// Mitsubishi GX Works2 project: BookEX6_IP102   PLC: Q06UDV

// global labels: Global
VAR_GLOBAL
  abArray0 AT M5010 : ARRAY [0..49] OF BOOL;
  sStr0 AT D5000 : STRING[199];
  sStr1 AT D5100 : STRING[199];
  sStr2 AT D5200 : STRING[199];
  sStr3 AT D5300 : STRING[199];
  sStr4 AT D5400 : STRING[199];
  sStr5 AT D5500 : STRING[199];
  sStr6 AT D5600 : STRING[199];
  sStr7 AT D5700 : STRING[199];
  sStr8 AT D5800 : STRING[199];
  sStr9 AT D5900 : STRING[199];
  iVar0 AT D4500 : INT;
  iVar1 AT D4501 : INT;
  iVar2 AT D4502 : INT;
  iVar3 AT D4503 : INT;
  iVar4 AT D4504 : INT;
  iVar5 AT D4505 : INT;
  iVar6 AT D4506 : INT;
  iVar7 AT D4507 : INT;
  iVar8 AT D4508 : INT;
  iVar9 AT D4509 : INT;
  dVar0 AT D4510 : DINT;
  dVar1 AT D4512 : DINT;
  dVar2 AT D4514 : DINT;
  dVar3 AT D4516 : DINT;
  dVar4 AT D4518 : DINT;
  dVar5 AT D4520 : DINT;
  dVar6 AT D4522 : DINT;
  dVar7 AT D4524 : DINT;
  dVar8 AT D4526 : DINT;
  dVar9 AT D4528 : DINT;
  wVar0 AT D4530 : WORD;
  wVar1 AT D4531 : WORD;
  wVar2 AT D4532 : WORD;
  wVar3 AT D4533 : WORD;
  wVar4 AT D4534 : WORD;
  wVar5 AT D4535 : WORD;
  wVar6 AT D4536 : WORD;
  wVar7 AT D4537 : WORD;
  wVar8 AT D4538 : WORD;
  wVar9 AT D4539 : WORD;
  dwVar0 AT D4540 : DWORD;
  dwVar1 AT D4542 : DWORD;
  dwVar2 AT D4544 : DWORD;
  dwVar3 AT D4546 : DWORD;
  dwVar4 AT D4548 : DWORD;
  dwVar5 AT D4550 : DWORD;
  dwVar6 AT D4552 : DWORD;
  dwVar7 AT D4554 : DWORD;
  dwVar8 AT D4556 : DWORD;
  dwVar9 AT D4558 : DWORD;
  fsVar0 AT D4560 : REAL;
  fsVar1 AT D4562 : REAL;
  fsVar2 AT D4564 : REAL;
  fsVar3 AT D4566 : REAL;
  fsVar4 AT D4568 : REAL;
  fsVar5 AT D4570 : REAL;
  fsVar6 AT D4572 : REAL;
  fsVar7 AT D4574 : REAL;
  fsVar8 AT D4576 : REAL;
  fsVar9 AT D4578 : REAL;
  fdVar0 AT D4580 : LREAL;
  tTime0 AT D4620 : TIME;
  tTime1 AT D4622 : TIME;
  tTime2 AT D4624 : TIME;
  tTime3 AT D4626 : TIME;
  tTime4 AT D4628 : TIME;
  tTime5 AT D4630 : TIME;
  tTime6 AT D4632 : TIME;
  tTime7 AT D4634 : TIME;
  tTime8 AT D4636 : TIME;
  tTime9 AT D4638 : TIME;
  tTime10 AT D4640 : TIME;
  bVar1 AT M5001 : BOOL;
  bVar2 AT M5002 : BOOL;
  bVar3 AT M5003 : BOOL;
  bVar4 AT M5004 : BOOL;
  bVar5 AT M5005 : BOOL;
  bVar6 AT M5006 : BOOL;
  bVar7 AT M5007 : BOOL;
  bVar8 AT M5008 : BOOL;
  bVar9 AT M5009 : BOOL;
  abArray1 AT M5060 : ARRAY [0..49] OF BOOL;
  abArray2 AT M5110 : ARRAY [0..49] OF BOOL;
  abArray3 AT M5160 : ARRAY [0..49] OF BOOL;
  abArray4 AT M5210 : ARRAY [0..49] OF BOOL;
  abArray5 AT M5260 : ARRAY [0..49] OF BOOL;
  abArray6 AT M5310 : ARRAY [0..49] OF BOOL;
  abArray7 AT M5360 : ARRAY [0..49] OF BOOL;
  abArray8 AT M5410 : ARRAY [0..49] OF BOOL;
  abArray9 AT M5460 : ARRAY [0..49] OF BOOL;
  fdVar1 AT D4584 : LREAL;
  fdVar2 AT D4588 : LREAL;
  fdVar3 AT D4592 : LREAL;
  fdVar4 AT D4596 : LREAL;
  fdVar5 AT D4600 : LREAL;
  fdVar6 AT D4604 : LREAL;
  fdVar7 AT D4608 : LREAL;
  fdVar8 AT D4612 : LREAL;
  fdVar9 AT D4616 : LREAL;
  bVar0 AT M5000 : BOOL;
END_VAR

// global labels: QPLCSpecial
VAR_GLOBAL
  sbGetTime AT SM213 : BOOL;
  sbOn AT SM400 : BOOL;
  sbOff AT SM401 : BOOL;
  sbOn1Time AT SM402 : BOOL;
  sbOff1Time AT SM403 : BOOL;
  sb5ms AT SM409 : BOOL;
  sdSwitch AT SD200 : INT;
  sdTime03 AT SD212 : INT;
  sdTime04 AT SD213 : INT;
  sdTime02 AT SD211 : INT;
  sdTime01 AT SD210 : INT;
  sdScanTime1 AT SD521 : INT;
  sdScanTimeMin1 AT SD525 : INT;
  sdScanTimeMin AT SD524 : INT;
  sdScanTimeMax1 AT SD527 : INT;
  sdScanTimeMax AT SD526 : INT;
  sbErrInfo2 AT SM16 : BOOL;
  sbErrInfo AT SM5 : BOOL;
  sbSelfError AT SM1 : BOOL;
  sbDiagError AT SM0 : BOOL;
  sbResetErr AT SM50 : BOOL;
  sbSetTime AT SM210 : BOOL;
  sbFuse AT SM60 : BOOL;
  sbOpError AT SM56 : BOOL;
  sbPowerDown AT SM53 : BOOL;
  sbBatLow AT SM52 : BOOL;
  sbBatLowL AT SM51 : BOOL;
  sbSTOP AT SM203 : BOOL;
  sbPAUSE AT SM204 : BOOL;
  sbNsec AT SM414 : BOOL;
  sb1000ms AT SM413 : BOOL;
  sb500ms AT SM412 : BOOL;
  sbNms AT SM415 : BOOL;
  sbUserClk4 AT SM424 : BOOL;
  sbUserClk3 AT SM423 : BOOL;
  sbUserClk2 AT SM422 : BOOL;
  sbUserClk1 AT SM421 : BOOL;
  sbUserClk0 AT SM420 : BOOL;
  sdBatLowL AT SD51 : INT;
  sdPLCErrInfo AT SD4 : INT;
  sdPLCErrDate2 AT SD3 : INT;
  sdPLCErrDate1 AT SD2 : INT;
  sdPLCErrDate0 AT SD1 : INT;
  sdPLCErrCode AT SD0 : INT;
  sdFuse AT SD60 : INT;
  sdPowerDown AT SD53 : INT;
  sdBatLow AT SD52 : INT;
  sdCPUSts AT SD203 : INT;
  sdLed AT SD201 : INT;
  sdScanTime AT SD520 : INT;
  sdCntNsec AT SD414 : INT;
  sdCnt1sec AT SD412 : INT;
  sdCntScan AT SD420 : INT;
  sdCntNms AT SD415 : INT;
  sb100ms AT SM411 : BOOL;
  sb50ms AT SM410 : BOOL;
  sdSckOpenComp AT SD1282 : WORD;
  sdSckOpenReq AT SD1284 : WORD;
  sdSckDataRx AT SD1286 : WORD;
  sdSckConn AT SD1288 : WORD;
END_VAR

// global labels: Network
VAR_GLOBAL
  aSendData1 AT D100 : ARRAY [0..4] OF INT;
  aiTxData AT D4000 : ARRAY [0..99] OF INT;
  aiRxData AT D4100 : ARRAY [0..99] OF INT;
  iOpenOK AT D3900 : INT;
  iOpenERR AT D3901 : INT;
  iSendOK AT D3902 : INT;
  iSendERR AT D3903 : INT;
  iCloseOK AT D3906 : INT;
  iCloseERR AT D3907 : INT;
  iRecvOK AT D3904 : INT;
  iRecvERR AT D3905 : INT;
  aiTxData2 AT D4200 : ARRAY [0..99] OF INT;
  aiRxData2 AT D4300 : ARRAY [0..99] OF INT;
  iOpenOK2 AT D3908 : INT;
  iOpenERR2 AT D3909 : INT;
  iSendOK2 AT D3910 : INT;
  iSendERR2 AT D3911 : INT;
  iRecvOK2 AT D3912 : INT;
  iRecvERR2 AT D3913 : INT;
  iCloseOK2 AT D3914 : INT;
  iCloseERR2 AT D3915 : INT;
  iEOpenComp AT D3916 : INT;
  iEOpenReq AT D3917 : INT;
  iERecvFlag AT D3918 : INT;
  iOpenCode AT D3919 : INT;
  iSendCode AT D3920 : INT;
  iRecvCode AT D3921 : INT;
  iCloseCode AT D3922 : INT;
  iOpenCode2 AT D3923 : INT;
  iSendCode2 AT D3924 : INT;
  iRecvCode2 AT D3925 : INT;
  iCloseCode2 AT D3926 : INT;
  aRecvData1 AT D105 : ARRAY [0..4] OF INT;
  aSendData2 AT D110 : ARRAY [0..4] OF INT;
  aRecvData2 AT D115 : ARRAY [0..4] OF INT;
  aSendData3 AT D120 : ARRAY [0..4] OF INT;
  aRecvData3 AT D125 : ARRAY [0..4] OF INT;
  aRdata AT D140 : ARRAY [0..9] OF INT;
  aSLMPDataTx AT D150 : ARRAY [0..9] OF WORD;
  aSLMPDataRx AT D160 : ARRAY [0..9] OF WORD;
END_VAR
// user libraries (not included): HMI

PROGRAM ExUINI
VAR
  bReq : BOOL;
  Mov8INT_1 : Mov8INT;
  abComp : ARRAY [0..1] OF BOOL;
  bNormal : BOOL;
  bError : BOOL;
END_VAR
(* structured ladder/FBD written out as ST: instructions are called as NAME(EN, inputs, outputs); _pN, _eN, _tN stand for wires *)
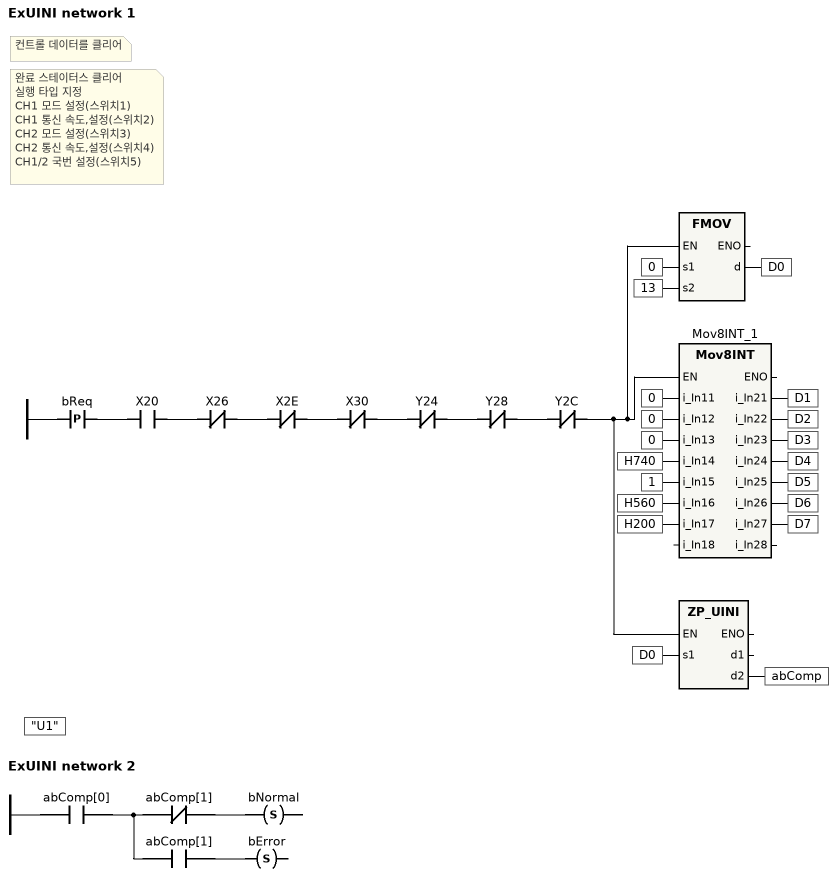
(* network 1 *)
(* 컨트롤 데이터를 클리어 *)
(* 완료 스테이터스 클리어 / 실행 타입 지정 / CH1 모드 설정(스위치1) / CH1 통신 속도,설정(스위치2) / CH2 모드 설정(스위치3) / CH2 통신 속도,설정(스위치4) / CH1/2 국번 설정(스위치5) *)
_p1 := LDP(TRUE, bReq) AND X20 AND NOT X26 AND NOT X2E AND NOT X30 AND NOT Y24 AND NOT Y28 AND NOT Y2C;
FMOV(_p1, 0, 13, D0);
Mov8INT_1(EN := _p1, i_In11 := 0, i_In12 := 0, i_In13 := 0, i_In14 := H740, i_In15 := 1, i_In16 := H560, i_In17 := H200, i_In21 => D1, i_In22 => D2, i_In23 => D3, i_In24 => D4, i_In25 => D5, i_In26 => D6, i_In27 => D7);
ZP_UINI(_p1, D0, _open, abComp);
(* not connected to any output: "U1" *)
(* network 2 *)
SET(abComp[0] AND NOT abComp[1], bNormal);
SET(abComp[0] AND abComp[1], bError);
END_PROGRAM

PROGRAM Ez_ethREAD_WRITE
VAR
  Mov8INT_1 : Mov8INT;
  acRdCtrl : ARRAY [0..17] OF INT;
  abRdComp : ARRAY [0..1] OF BOOL;
  iCntRdOk : INT;
  iCntRdErr : INT;
END_VAR
(* structured ladder/FBD written out as ST: instructions are called as NAME(EN, inputs, outputs); _pN, _eN, _tN stand for wires *)
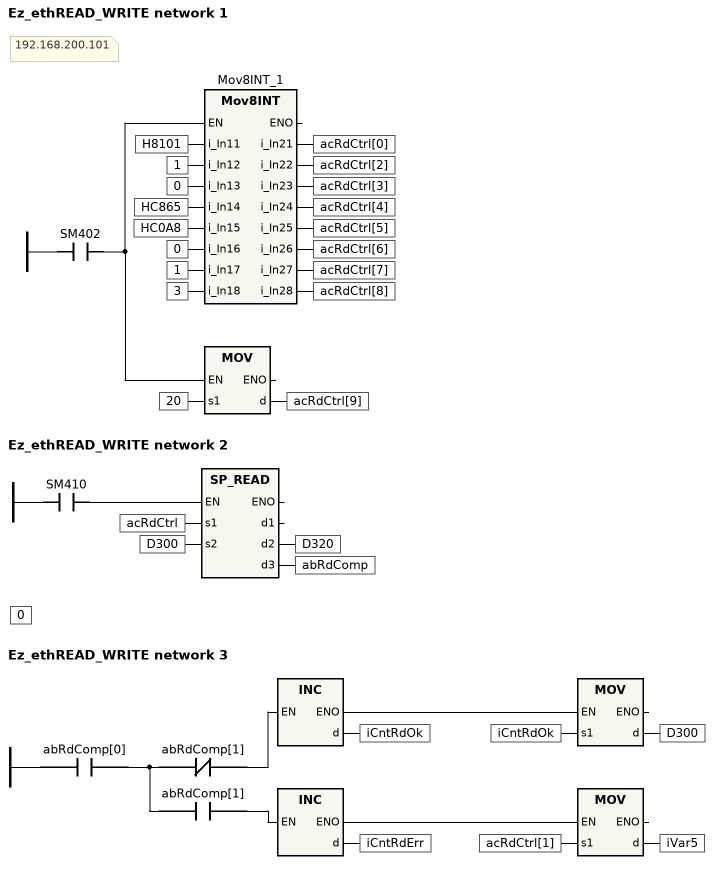
(* network 1 *)
(* 192.168.200.101 *)
Mov8INT_1(EN := SM402, i_In11 := H8101, i_In12 := 1, i_In13 := 0, i_In14 := HC865, i_In15 := HC0A8, i_In16 := 0, i_In17 := 1, i_In18 := 3, i_In21 => acRdCtrl[0], i_In22 => acRdCtrl[2], i_In23 => acRdCtrl[3], i_In24 => acRdCtrl[4], i_In25 => acRdCtrl[5], i_In26 => acRdCtrl[6], i_In27 => acRdCtrl[7], i_In28 => acRdCtrl[8]);
MOV(SM402, 20, acRdCtrl[9]);
(* network 2 *)
SP_READ(SM410, acRdCtrl, D300, _open, D320, abRdComp);
(* not connected to any output: 0 *)
(* network 3 *)
_e1 := INC(abRdComp[0] AND NOT abRdComp[1], iCntRdOk);
MOV(_e1, iCntRdOk, D300);
_e2 := INC(abRdComp[0] AND abRdComp[1], iCntRdErr);
MOV(_e2, acRdCtrl[1], iVar5);
END_PROGRAM

PROGRAM ExSample
VAR
  Mov8INT_1 : Mov8INT;
  Mov8INT_2 : Mov8INT;
  Mov8INT_3 : Mov8INT;
  Mov8INT_4 : Mov8INT;
  Mov8INT_5 : Mov8INT;
  Mov8INT_6 : Mov8INT;
END_VAR
(* structured ladder/FBD written out as ST: instructions are called as NAME(EN, inputs, outputs); _pN, _eN, _tN stand for wires *)
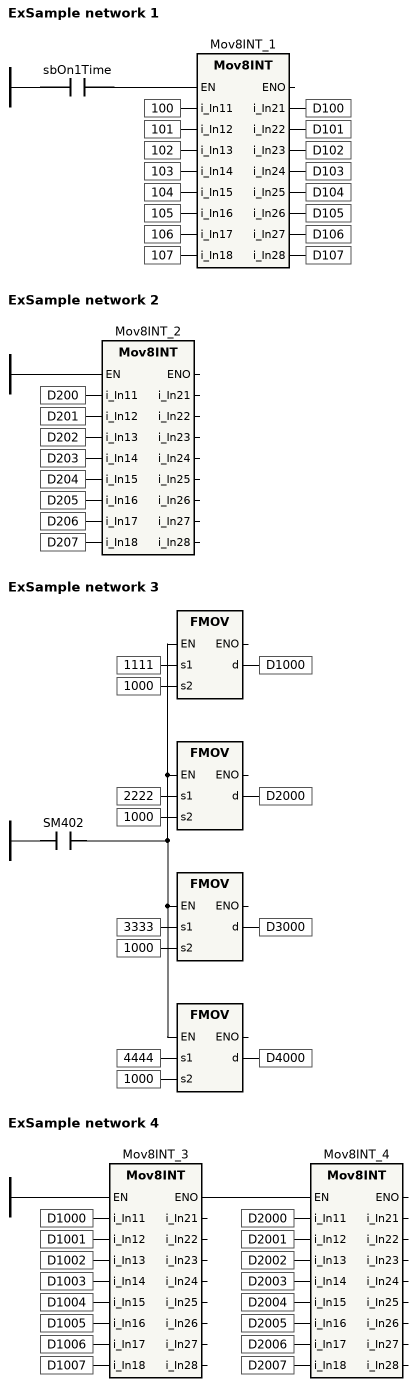
(* network 1 *)
Mov8INT_1(EN := sbOn1Time, i_In11 := 100, i_In12 := 101, i_In13 := 102, i_In14 := 103, i_In15 := 104, i_In16 := 105, i_In17 := 106, i_In18 := 107, i_In21 => D100, i_In22 => D101, i_In23 => D102, i_In24 => D103, i_In25 => D104, i_In26 => D105, i_In27 => D106, i_In28 => D107);
(* network 2 *)
Mov8INT_2(EN := TRUE, i_In11 := D200, i_In12 := D201, i_In13 := D202, i_In14 := D203, i_In15 := D204, i_In16 := D205, i_In17 := D206, i_In18 := D207);
(* network 3 *)
FMOV(SM402, 1111, 1000, D1000);
FMOV(SM402, 2222, 1000, D2000);
FMOV(SM402, 3333, 1000, D3000);
FMOV(SM402, 4444, 1000, D4000);
(* network 4 *)
Mov8INT_3(EN := TRUE, i_In11 := D1000, i_In12 := D1001, i_In13 := D1002, i_In14 := D1003, i_In15 := D1004, i_In16 := D1005, i_In17 := D1006, i_In18 := D1007);
Mov8INT_4(EN := Mov8INT_3.ENO, i_In11 := D2000, i_In12 := D2001, i_In13 := D2002, i_In14 := D2003, i_In15 := D2004, i_In16 := D2005, i_In17 := D2006, i_In18 := D2007);
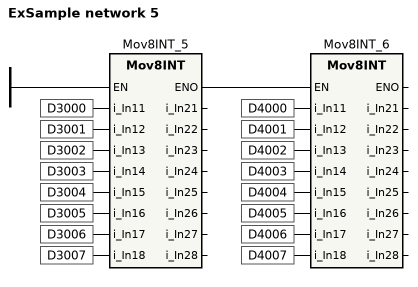
(* network 5 *)
Mov8INT_5(EN := TRUE, i_In11 := D3000, i_In12 := D3001, i_In13 := D3002, i_In14 := D3003, i_In15 := D3004, i_In16 := D3005, i_In17 := D3006, i_In18 := D3007);
Mov8INT_6(EN := Mov8INT_5.ENO, i_In11 := D4000, i_In12 := D4001, i_In13 := D4002, i_In14 := D4003, i_In15 := D4004, i_In16 := D4005, i_In17 := D4006, i_In18 := D4007);
END_PROGRAM

PROGRAM ExMBRW
VAR
  bReq : BOOL;
  acData : ARRAY [0..16] OF INT;
  Mov8INT_1 : Mov8INT;
  Mov8INT_2 : Mov8INT;
  abRes : ARRAY [0..1] OF BOOL;
  bOK : BOOL;
  bERR : BOOL;
  ErrCode : INT;
  Mov8INT_3 : Mov8INT;
  Mov4INT_1 : Mov4INT;
END_VAR
(* structured ladder/FBD written out as ST: instructions are called as NAME(EN, inputs, outputs); _pN, _eN, _tN stand for wires *)
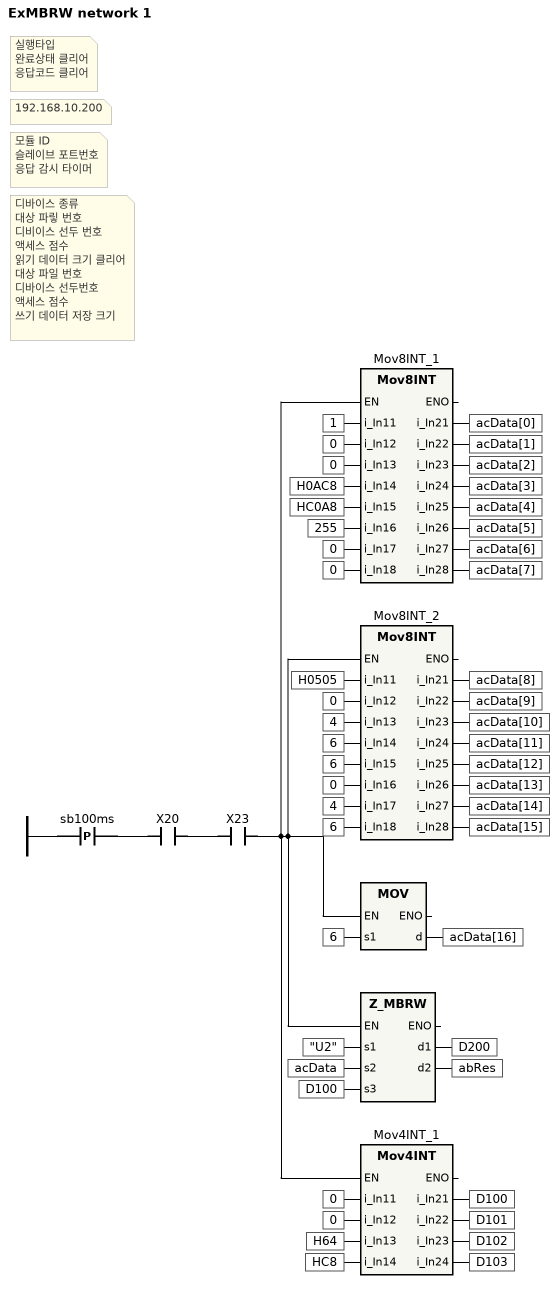
(* network 1 *)
(* 실행타입 / 완료상태 클리어 / 응답코드 클리어 *)
(* 192.168.10.200 *)
(* 모듈 ID / 슬레이브 포트번호 / 응답 감시 타이머 *)
(* 디바이스 종류 / 대상 파맇 번호 / 디비이스 선두 번호 / 액세스 점수 / 읽기 데이터 크기 클리어 / 대상 파일 번호 / 디바이스 선두번호 / 액세스 점수 / 쓰기 데이터 저장 크기 *)
_p1 := LDP(TRUE, sb100ms) AND X20 AND X23;
Mov8INT_1(EN := _p1, i_In11 := 1, i_In12 := 0, i_In13 := 0, i_In14 := H0AC8, i_In15 := HC0A8, i_In16 := 255, i_In17 := 0, i_In18 := 0, i_In21 => acData[0], i_In22 => acData[1], i_In23 => acData[2], i_In24 => acData[3], i_In25 => acData[4], i_In26 => acData[5], i_In27 => acData[6], i_In28 => acData[7]);
Mov8INT_2(EN := _p1, i_In11 := H0505, i_In12 := 0, i_In13 := 4, i_In14 := 6, i_In15 := 6, i_In16 := 0, i_In17 := 4, i_In18 := 6, i_In21 => acData[8], i_In22 => acData[9], i_In23 => acData[10], i_In24 => acData[11], i_In25 => acData[12], i_In26 => acData[13], i_In27 => acData[14], i_In28 => acData[15]);
MOV(_p1, 6, acData[16]);
Z_MBRW(_p1, "U2", acData, D100, D200, abRes);
Mov4INT_1(EN := _p1, i_In11 := 0, i_In12 := 0, i_In13 := H64, i_In14 := HC8, i_In21 => D100, i_In22 => D101, i_In23 => D102, i_In24 => D103);
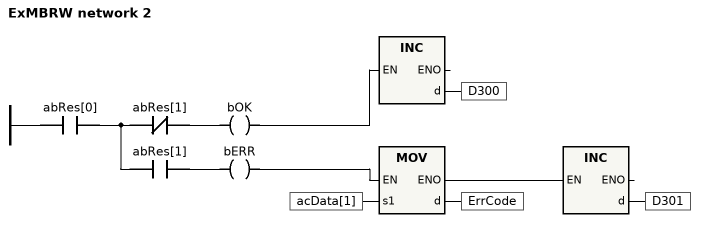
(* network 2 *)
_p1 := abRes[0] AND NOT abRes[1];
bOK := _p1;
INC(_p1, D300);
_p2 := abRes[0] AND abRes[1];
bERR := _p2;
_e3 := MOV(_p2, acData[1], ErrCode);
INC(_e3, D301);
END_PROGRAM

PROGRAM ExMBREQ
VAR
  Req : BOOL;
  acData : ARRAY [0..7] OF INT;
  Mov8INT_1 : Mov8INT;
  Mov8INT_2 : Mov8INT;
  abRes : ARRAY [0..1] OF BOOL;
  bOK : BOOL;
  bERR : BOOL;
  ErrCode : INT;
  bReqOFF : BOOL;
  bReqPing : BOOL;
  bReqSend : BOOL;
  Mov4INT_1 : Mov4INT;
  Mov4INT_2 : Mov4INT;
END_VAR
(* structured ladder/FBD written out as ST: instructions are called as NAME(EN, inputs, outputs); _pN, _eN, _tN stand for wires *)
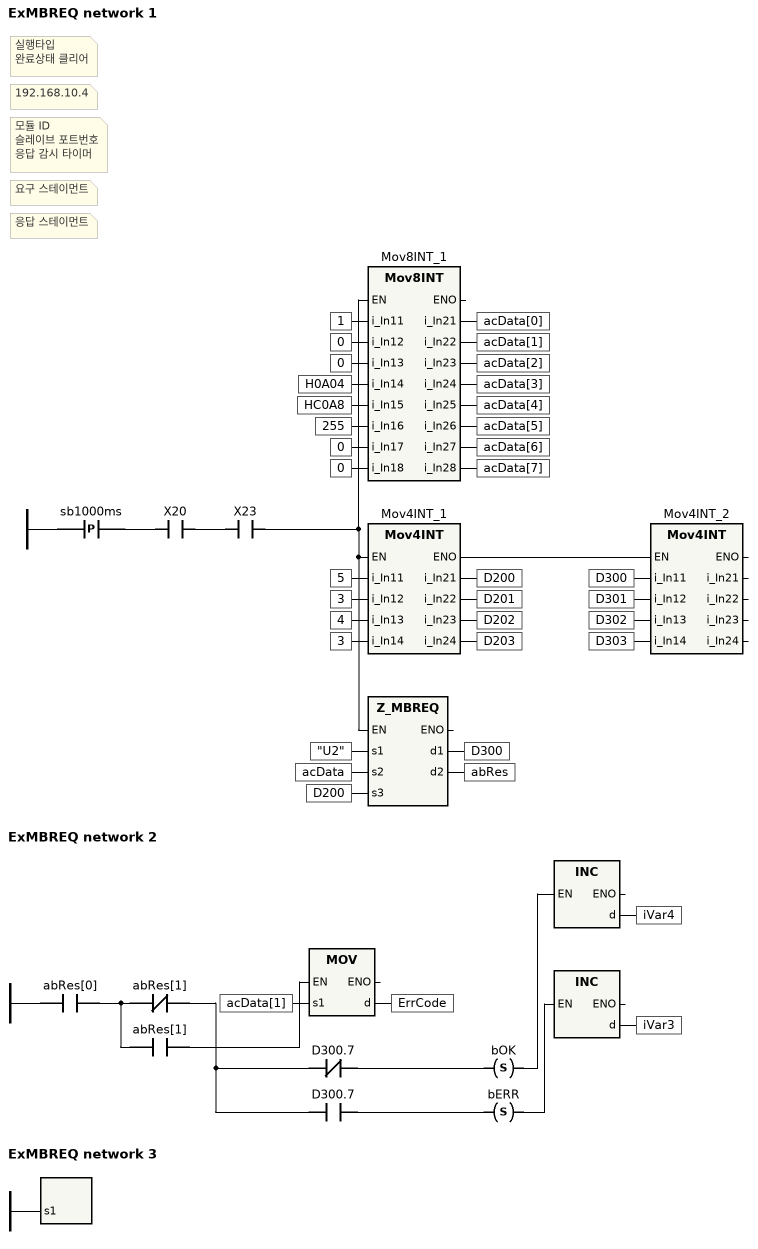
(* network 1 *)
(* 실행타입 / 완료상태 클리어 *)
(* 192.168.10.4 *)
(* 모듈 ID / 슬레이브 포트번호 / 응답 감시 타이머 *)
(* 요구 스테이먼트 *)
(* 응답 스테이먼트 *)
_p1 := LDP(TRUE, sb1000ms) AND X20 AND X23;
Mov8INT_1(EN := _p1, i_In11 := 1, i_In12 := 0, i_In13 := 0, i_In14 := H0A04, i_In15 := HC0A8, i_In16 := 255, i_In17 := 0, i_In18 := 0, i_In21 => acData[0], i_In22 => acData[1], i_In23 => acData[2], i_In24 => acData[3], i_In25 => acData[4], i_In26 => acData[5], i_In27 => acData[6], i_In28 => acData[7]);
Mov4INT_1(EN := _p1, i_In11 := 5, i_In12 := 3, i_In13 := 4, i_In14 := 3, i_In21 => D200, i_In22 => D201, i_In23 => D202, i_In24 => D203);
Mov4INT_2(EN := Mov4INT_1.ENO, i_In11 := D300, i_In12 := D301, i_In13 := D302, i_In14 := D303);
Z_MBREQ(_p1, "U2", acData, D200, D300, abRes);
(* network 2 *)
_p1 := abRes[0] AND NOT abRes[1];
_p2 := _p1 AND NOT D300.7;
SET(_p2, bOK);
INC(_p2, iVar4);
_p3 := _p1 AND D300.7;
SET(_p3, bERR);
INC(_p3, iVar3);
MOV(abRes[0] AND abRes[1], acData[1], ErrCode);
(* network 3 *)
(* element kind 10  <- TRUE *)
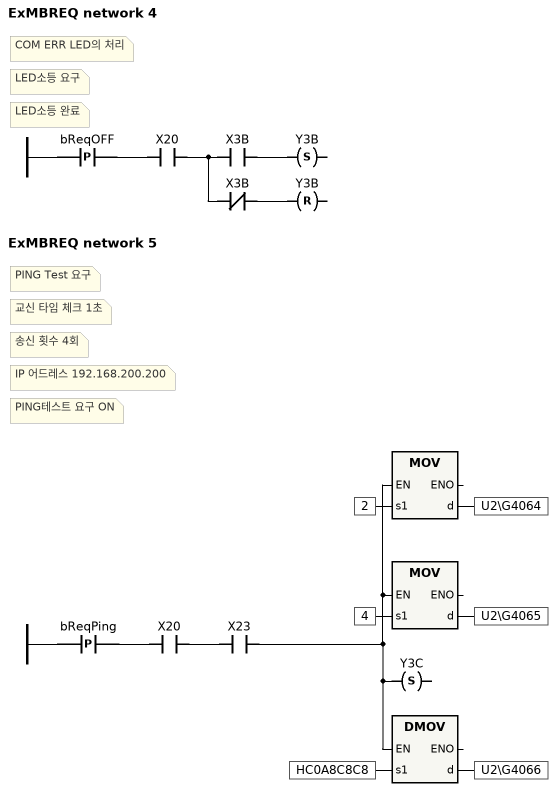
(* network 4 *)
(* COM ERR LED의 처리 *)
(* LED소등 요구 *)
(* LED소등 완료 *)
_p1 := LDP(TRUE, bReqOFF) AND X20;
SET(_p1 AND X3B, Y3B);
RST(_p1 AND NOT X3B, Y3B);
(* network 5 *)
(* PING Test 요구 *)
(* 교신 타임 체크 1초 *)
(* 송신 횟수 4회 *)
(* IP 어드레스 192.168.200.200 *)
(* PING테스트 요구 ON *)
_p1 := LDP(TRUE, bReqPing) AND X20 AND X23;
MOV(_p1, 2, U2\G4064);
MOV(_p1, 4, U2\G4065);
DMOV(_p1, HC0A8C8C8, U2\G4066);
SET(_p1, Y3C);
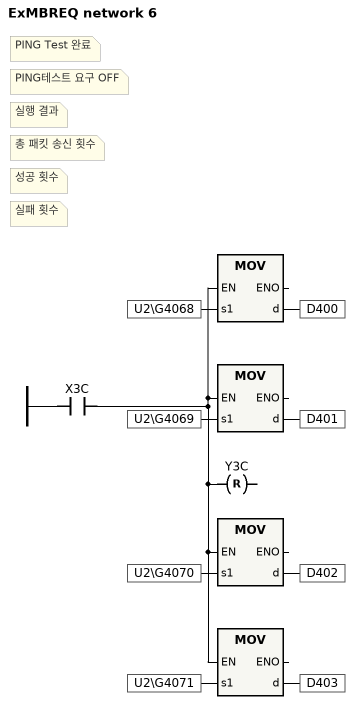
(* network 6 *)
(* PING Test 완료 *)
(* PING테스트 요구 OFF *)
(* 실행 결과 *)
(* 총 패킷 송신 횟수 *)
(* 성공 횟수 *)
(* 실패 횟수 *)
RST(X3C, Y3C);
MOV(X3C, U2\G4068, D400);
MOV(X3C, U2\G4069, D401);
MOV(X3C, U2\G4070, D402);
MOV(X3C, U2\G4071, D403);
END_PROGRAM

PROGRAM Ex_SewData6
VAR
  bOpenReqC : BOOL;
  bCsetReq : BOOL;
  bOpenReqE : BOOL;
  bOpenOkC : BOOL;
  bOpenOkE : BOOL;
  bOpenErrC : BOOL;
  bOpenErrE : BOOL;
  abOpenResC : ARRAY [0..1] OF BOOL;
  abOpenResE : ARRAY [0..1] OF BOOL;
  acOpenData : ARRAY [0..9] OF INT;
  acCsetData : ARRAY [0..4] OF INT;
  acRdCtrl : ARRAY [0..9] OF INT;
  bSendReqC : BOOL;
  bSendReqE : BOOL;
  bSendOkC : BOOL;
  bSendOkE : BOOL;
  bSendErrC : BOOL;
  bSendErrE : BOOL;
  abSendResC : ARRAY [0..1] OF BOOL;
  abSendResE : ARRAY [0..1] OF BOOL;
  abSendResF : ARRAY [0..1] OF BOOL;
  acSendDataC : ARRAY [0..1] OF INT;
  acSendDataE : ARRAY [0..1] OF INT;
  acSendDataF : ARRAY [0..1] OF INT;
  bRecvOkC : BOOL;
  bRecvOkE : BOOL;
  bRecvOkF : BOOL;
  bRecvErrC : BOOL;
  bRecvErrE : BOOL;
  bRecvErrF : BOOL;
  abRecvResC : ARRAY [0..1] OF BOOL;
  abRecvResE : ARRAY [0..1] OF BOOL;
  abRecvResF : ARRAY [0..1] OF BOOL;
  acRecvDataC : ARRAY [0..1] OF INT;
  acRecvDataE : ARRAY [0..1] OF INT;
  acRecvDataF : ARRAY [0..1] OF INT;
  bCloseReq : BOOL;
  bCloseOkC : BOOL;
  bCloseOkE : BOOL;
  bCloseErrC : BOOL;
  bCloseErrE : BOOL;
  abCloseResC : ARRAY [0..1] OF BOOL;
  abCloseResE : ARRAY [0..1] OF BOOL;
  acCloseData : ARRAY [0..1] OF INT;
  CntSend1 : INT;
  CntSend2 : INT;
  CntSend3 : INT;
  CntRecv1 : INT;
  CntRecvErr1 : INT;
  CntRecv2 : INT;
  CntRecv3 : INT;
  CntRecvErr2 : INT;
  CntRecvErr3 : INT;
  ErrCodeSC : INT;
  ErrCodeSE : INT;
  ErrCodeSF : INT;
  ErrCodeRC : INT;
  ErrCodeRE : INT;
  ErrCodeRF : INT;
  Mov4INT_1 : Mov4INT;
  Mov8INT_1 : Mov8INT;
  Mov4INT_2 : Mov4INT;
  Mov4INT_3 : Mov4INT;
  Mov4INT_4 : Mov4INT;
  Word2Bit8_1 : Word2Bit8;
  Word2Bit8_2 : Word2Bit8;
  Word2Bit8_3 : Word2Bit8;
  Word2Bit8_4 : Word2Bit8;
  Word2Bit8_5 : Word2Bit8;
  Word2Bit8_6 : Word2Bit8;
  TON_1 : TON;
  TON_2 : TON;
  TON_3 : TON;
  sbTxReq : BOOL;
  Mov4INT_5 : Mov4INT;
  Mov8INT_2 : Mov8INT;
  Mov8INT_3 : Mov8INT;
  Mov8INT_4 : Mov8INT;
  Mov8INT_5 : Mov8INT;
  TxSet : BOOL;
  TxReq : BOOL;
END_VAR
(* structured ladder/FBD written out as ST: instructions are called as NAME(EN, inputs, outputs); _pN, _eN, _tN stand for wires *)
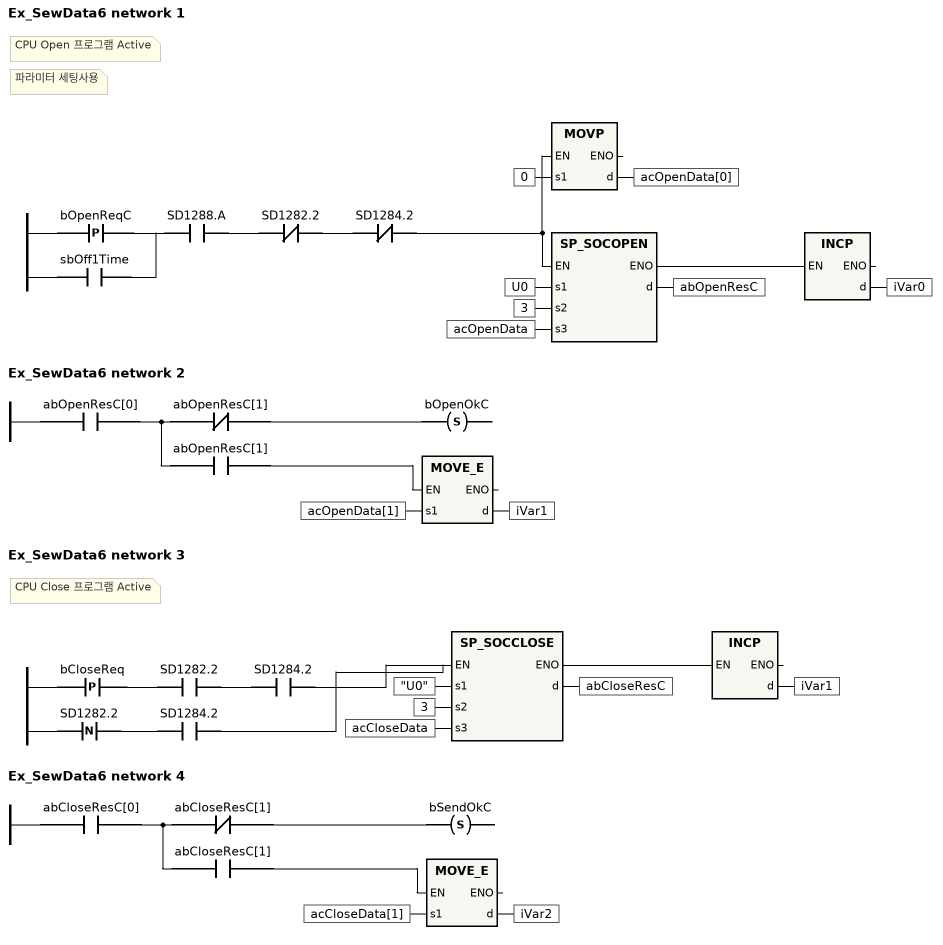
(* network 1 *)
(* CPU Open 프로그램 Active *)
(* 파라미터 세팅사용 *)
_p1 := (((LDP(TRUE, bOpenReqC) OR sbOff1Time) AND SD1288.A) AND NOT SD1282.2) AND NOT SD1284.2;
MOVP(_p1, 0, acOpenData[0]);
_e2 := SP_SOCOPEN(_p1, U0, 3, acOpenData, abOpenResC);
INCP(_e2, iVar0);
(* network 2 *)
SET(abOpenResC[0] AND NOT abOpenResC[1], bOpenOkC);
MOVE_E(abOpenResC[0] AND abOpenResC[1], acOpenData[1], iVar1);
(* network 3 *)
(* CPU Close 프로그램 Active *)
_e1 := SP_SOCCLOSE((LDP(TRUE, bCloseReq) AND SD1282.2 AND SD1284.2) OR (LDF(TRUE, SD1282.2) AND SD1284.2), "U0", 3, acCloseData, abCloseResC);
INCP(_e1, iVar1);
(* network 4 *)
SET(abCloseResC[0] AND NOT abCloseResC[1], bSendOkC);
MOVE_E(abCloseResC[0] AND abCloseResC[1], acCloseData[1], iVar2);
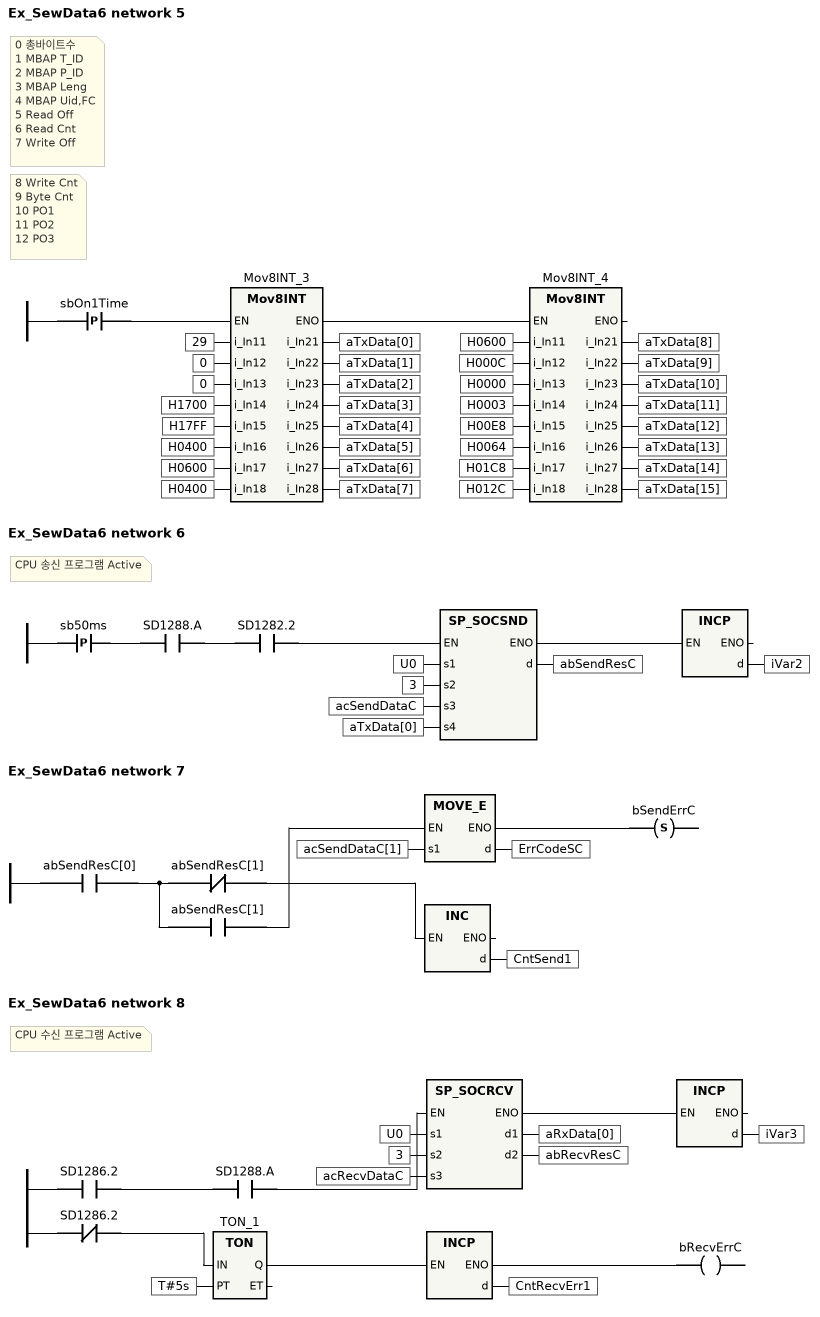
(* network 5 *)
(* 0 총바이트수 / 1 MBAP T_ID / 2 MBAP P_ID / 3 MBAP Leng / 4 MBAP Uid,FC / 5 Read Off / 6 Read Cnt / 7 Write Off *)
(* 8 Write Cnt / 9 Byte Cnt  / 10 PO1 / 11 PO2 / 12 PO3 *)
Mov8INT_3(EN := LDP(TRUE, sbOn1Time), i_In11 := 29, i_In12 := 0, i_In13 := 0, i_In14 := H1700, i_In15 := H17FF, i_In16 := H0400, i_In17 := H0600, i_In18 := H0400, i_In21 => aTxData[0], i_In22 => aTxData[1], i_In23 => aTxData[2], i_In24 => aTxData[3], i_In25 => aTxData[4], i_In26 => aTxData[5], i_In27 => aTxData[6], i_In28 => aTxData[7]);
Mov8INT_4(EN := Mov8INT_3.ENO, i_In11 := H0600, i_In12 := H000C, i_In13 := H0000, i_In14 := H0003, i_In15 := H00E8, i_In16 := H0064, i_In17 := H01C8, i_In18 := H012C, i_In21 => aTxData[8], i_In22 => aTxData[9], i_In23 => aTxData[10], i_In24 => aTxData[11], i_In25 => aTxData[12], i_In26 => aTxData[13], i_In27 => aTxData[14], i_In28 => aTxData[15]);
(* network 6 *)
(* CPU 송신 프로그램 Active *)
_e1 := SP_SOCSND(LDP(TRUE, sb50ms) AND SD1288.A AND SD1282.2, U0, 3, acSendDataC, aTxData[0], abSendResC);
INCP(_e1, iVar2);
(* network 7 *)
INC(abSendResC[0] AND NOT abSendResC[1], CntSend1);
_e1 := MOVE_E(abSendResC[0] AND abSendResC[1], acSendDataC[1], ErrCodeSC);
SET(_e1, bSendErrC);
(* network 8 *)
(* CPU 수신 프로그램 Active *)
_e1 := SP_SOCRCV(SD1286.2 AND SD1288.A, U0, 3, acRecvDataC, aRxData[0], abRecvResC);
INCP(_e1, iVar3);
TON_1(IN := NOT SD1286.2, PT := T#5s);
_e2 := INCP(TON_1.Q, CntRecvErr1);
bRecvErrC := _e2;
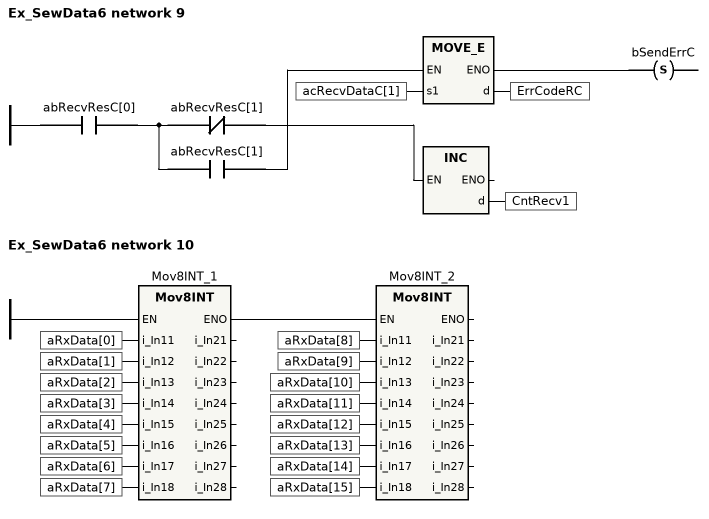
(* network 9 *)
INC(abRecvResC[0] AND NOT abRecvResC[1], CntRecv1);
_e1 := MOVE_E(abRecvResC[0] AND abRecvResC[1], acRecvDataC[1], ErrCodeRC);
SET(_e1, bSendErrC);
(* network 10 *)
Mov8INT_1(EN := TRUE, i_In11 := aRxData[0], i_In12 := aRxData[1], i_In13 := aRxData[2], i_In14 := aRxData[3], i_In15 := aRxData[4], i_In16 := aRxData[5], i_In17 := aRxData[6], i_In18 := aRxData[7]);
Mov8INT_2(EN := Mov8INT_1.ENO, i_In11 := aRxData[8], i_In12 := aRxData[9], i_In13 := aRxData[10], i_In14 := aRxData[11], i_In15 := aRxData[12], i_In16 := aRxData[13], i_In17 := aRxData[14], i_In18 := aRxData[15]);
END_PROGRAM

FUNCTION_BLOCK Word2Bit16
VAR_INPUT
  bEN : BOOL;
END_VAR
VAR_OUTPUT
  Bit0 : BOOL;
  Bit1 : BOOL;
  Bit2 : BOOL;
  Bit3 : BOOL;
  Bit4 : BOOL;
  Bit5 : BOOL;
  Bit6 : BOOL;
  Bit7 : BOOL;
  Bit8 : BOOL;
  Bit9 : BOOL;
  Bit10 : BOOL;
  Bit11 : BOOL;
  Bit12 : BOOL;
  Bit13 : BOOL;
  Bit14 : BOOL;
  Bit15 : BOOL;
END_VAR
VAR_INPUT
  InWord : WORD;
END_VAR
VAR_OUTPUT
  bENO : BOOL;
END_VAR
VAR
  InVal : WORD;
END_VAR
 
bENO := bEN;
InVal :=InWord;
Bit0 := (InVal AND 16#0001) = H0001;
Bit1 := (InVal AND 16#0002) = H0002;
Bit2 := (InVal AND 16#0004) = H0004;
Bit3 := (InVal AND 16#0008) = H0008;
Bit4 := (InVal AND 16#0010) = H0010;
Bit5 := (InVal AND 16#0020) = H0020;
Bit6 := (InVal AND 16#0040) = H0040;
Bit7 := (InVal AND 16#0080) = H0080;
Bit8 := (InVal AND 16#0100) = H0100;
Bit9 := (InVal AND 16#0200) = H0200;
Bit10 := (InVal AND 16#0400) = H0400;
Bit11 := (InVal AND 16#0800) = H0800;
Bit12 := (InVal AND 16#1000) = H1000;
Bit13 := (InVal AND 16#2000) = H2000;
Bit14 := (InVal AND 16#4000) = H4000;
Bit15 := (InVal AND 16#8000) = H8000;

(*
Bit0 := WORD_TO_BOOL(IN AND 16#0001);
Bit1 := WORD_TO_BOOL(SHR(IN AND 16#0002 , 1));
Bit2 := WORD_TO_BOOL(SHR(IN AND 16#0004 , 2));
Bit3 := WORD_TO_BOOL(SHR(IN AND 16#0008 , 3));
Bit4 := WORD_TO_BOOL(SHR(IN AND 16#0010 , 4));
Bit5 := WORD_TO_BOOL(SHR(IN AND 16#0020 , 5));
Bit6 := WORD_TO_BOOL(SHR(IN AND 16#0040 , 6));
Bit7 := WORD_TO_BOOL(SHR(IN AND 16#0080 , 7));
 
Bit8 := WORD_TO_BOOL(SHR(IN AND 16#0100 , 8));
Bit9 := WORD_TO_BOOL(SHR(IN AND 16#0200 , 9));
Bit10 := WORD_TO_BOOL(SHR(IN AND 16#0400 , 10));
Bit11 := WORD_TO_BOOL(SHR(IN AND 16#0800 , 11));
Bit12 := WORD_TO_BOOL(SHR(IN AND 16#1000 , 12));
Bit13 := WORD_TO_BOOL(SHR(IN AND 16#2000 , 13));
Bit14 := WORD_TO_BOOL(SHR(IN AND 16#4000 , 14));
Bit15 := WORD_TO_BOOL(SHR(IN AND 16#8000 , 15));
*)
END_FUNCTION_BLOCK

FUNCTION_BLOCK Word2Bit8
VAR_INPUT
  IN : WORD;
END_VAR
VAR_OUTPUT
  Bit0 : BOOL;
  Bit1 : BOOL;
  Bit2 : BOOL;
  Bit3 : BOOL;
  Bit4 : BOOL;
  Bit5 : BOOL;
  Bit6 : BOOL;
  Bit7 : BOOL;
END_VAR
 
Bit0 := WORD_TO_BOOL(IN AND 16#0001);
Bit1 := WORD_TO_BOOL(SHR(IN AND 16#0002 , 1));
Bit2 := WORD_TO_BOOL(SHR(IN AND 16#0004 , 2));
Bit3 := WORD_TO_BOOL(SHR(IN AND 16#0008 , 3));
Bit4 := WORD_TO_BOOL(SHR(IN AND 16#0010 , 4));
Bit5 := WORD_TO_BOOL(SHR(IN AND 16#0020 , 5));
Bit6 := WORD_TO_BOOL(SHR(IN AND 16#0040 , 6));
Bit7 := WORD_TO_BOOL(SHR(IN AND 16#0080 , 7));
END_FUNCTION_BLOCK

PROGRAM Ex_SewData3
VAR
  bOpenReqC : BOOL;
  bCsetReq : BOOL;
  bOpenReqE : BOOL;
  bOpenOkC : BOOL;
  bOpenOkE : BOOL;
  bOpenErrC : BOOL;
  bOpenErrE : BOOL;
  abOpenResC : ARRAY [0..1] OF BOOL;
  abOpenResE : ARRAY [0..1] OF BOOL;
  acOpenData : ARRAY [0..9] OF INT;
  acCsetData : ARRAY [0..4] OF INT;
  acRdCtrl : ARRAY [0..9] OF INT;
  bSendReqC : BOOL;
  bSendReqE : BOOL;
  bSendOkC : BOOL;
  bSendOkE : BOOL;
  bSendErrC : BOOL;
  bSendErrE : BOOL;
  abSendResC : ARRAY [0..1] OF BOOL;
  abSendResE : ARRAY [0..1] OF BOOL;
  abSendResF : ARRAY [0..1] OF BOOL;
  acSendDataC : ARRAY [0..1] OF INT;
  acSendDataE : ARRAY [0..1] OF INT;
  acSendDataF : ARRAY [0..1] OF INT;
  bRecvOkC : BOOL;
  bRecvOkE : BOOL;
  bRecvOkF : BOOL;
  bRecvErrC : BOOL;
  bRecvErrE : BOOL;
  bRecvErrF : BOOL;
  abRecvResC : ARRAY [0..1] OF BOOL;
  abRecvResE : ARRAY [0..1] OF BOOL;
  abRecvResF : ARRAY [0..1] OF BOOL;
  acRecvDataC : ARRAY [0..1] OF INT;
  acRecvDataE : ARRAY [0..1] OF INT;
  acRecvDataF : ARRAY [0..1] OF INT;
  bCloseReq : BOOL;
  bCloseOkC : BOOL;
  bCloseOkE : BOOL;
  bCloseErrC : BOOL;
  bCloseErrE : BOOL;
  abCloseResC : ARRAY [0..1] OF BOOL;
  abCloseResE : ARRAY [0..1] OF BOOL;
  acCloseData : ARRAY [0..1] OF INT;
  CntSend1 : INT;
  CntSend2 : INT;
  CntSend3 : INT;
  CntRecv1 : INT;
  CntRecvErr1 : INT;
  CntRecv2 : INT;
  CntRecv3 : INT;
  CntRecvErr2 : INT;
  CntRecvErr3 : INT;
  ErrCodeSC : INT;
  ErrCodeSE : INT;
  ErrCodeSF : INT;
  ErrCodeRC : INT;
  ErrCodeRE : INT;
  ErrCodeRF : INT;
  Mov4INT_1 : Mov4INT;
  Mov8INT_1 : Mov8INT;
  Mov4INT_2 : Mov4INT;
  Mov4INT_3 : Mov4INT;
  Mov4INT_4 : Mov4INT;
  Word2Bit8_1 : Word2Bit8;
  Word2Bit8_2 : Word2Bit8;
  Word2Bit8_3 : Word2Bit8;
  Word2Bit8_4 : Word2Bit8;
  Word2Bit8_5 : Word2Bit8;
  Word2Bit8_6 : Word2Bit8;
  TON_1 : TON;
  TON_2 : TON;
  TON_3 : TON;
  sbTxReq : BOOL;
  Mov4INT_5 : Mov4INT;
  Mov8INT_2 : Mov8INT;
  Mov8INT_3 : Mov8INT;
  Mov8INT_4 : Mov8INT;
  Mov8INT_5 : Mov8INT;
  TxSet : BOOL;
  TxReq : BOOL;
END_VAR
(* structured ladder/FBD written out as ST: instructions are called as NAME(EN, inputs, outputs); _pN, _eN, _tN stand for wires *)
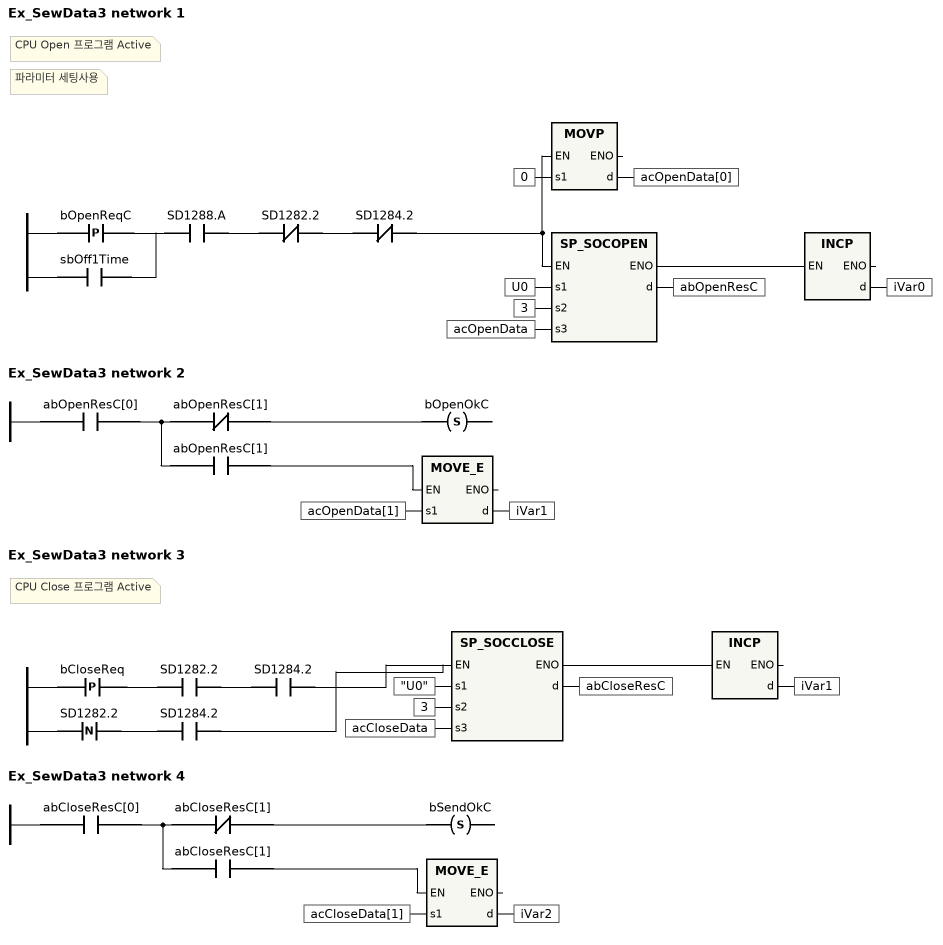
(* network 1 *)
(* CPU Open 프로그램 Active *)
(* 파라미터 세팅사용 *)
_p1 := (((LDP(TRUE, bOpenReqC) OR sbOff1Time) AND SD1288.A) AND NOT SD1282.2) AND NOT SD1284.2;
MOVP(_p1, 0, acOpenData[0]);
_e2 := SP_SOCOPEN(_p1, U0, 3, acOpenData, abOpenResC);
INCP(_e2, iVar0);
(* network 2 *)
SET(abOpenResC[0] AND NOT abOpenResC[1], bOpenOkC);
MOVE_E(abOpenResC[0] AND abOpenResC[1], acOpenData[1], iVar1);
(* network 3 *)
(* CPU Close 프로그램 Active *)
_e1 := SP_SOCCLOSE((LDP(TRUE, bCloseReq) AND SD1282.2 AND SD1284.2) OR (LDF(TRUE, SD1282.2) AND SD1284.2), "U0", 3, acCloseData, abCloseResC);
INCP(_e1, iVar1);
(* network 4 *)
SET(abCloseResC[0] AND NOT abCloseResC[1], bSendOkC);
MOVE_E(abCloseResC[0] AND abCloseResC[1], acCloseData[1], iVar2);
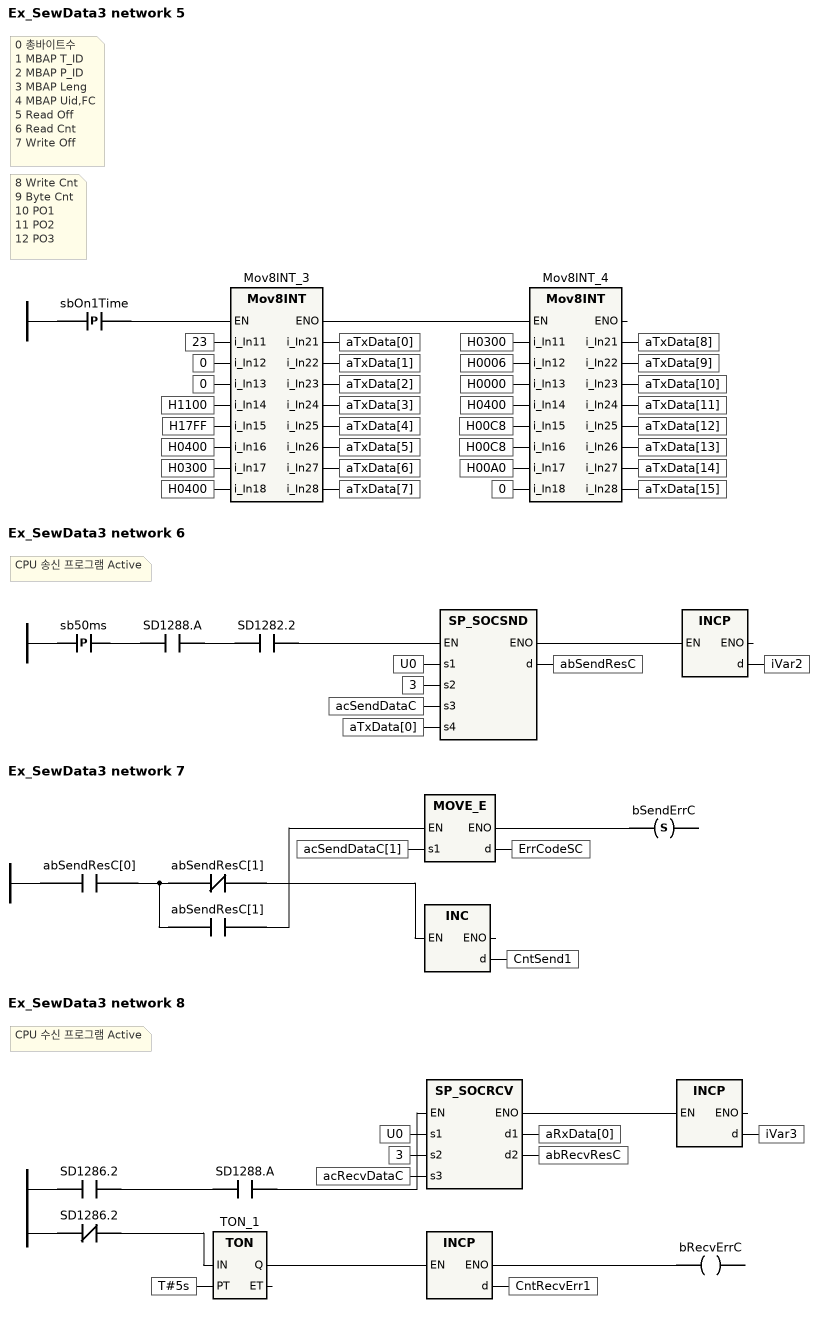
(* network 5 *)
(* 0 총바이트수 / 1 MBAP T_ID / 2 MBAP P_ID / 3 MBAP Leng / 4 MBAP Uid,FC / 5 Read Off / 6 Read Cnt / 7 Write Off *)
(* 8 Write Cnt / 9 Byte Cnt  / 10 PO1 / 11 PO2 / 12 PO3 *)
Mov8INT_3(EN := LDP(TRUE, sbOn1Time), i_In11 := 23, i_In12 := 0, i_In13 := 0, i_In14 := H1100, i_In15 := H17FF, i_In16 := H0400, i_In17 := H0300, i_In18 := H0400, i_In21 => aTxData[0], i_In22 => aTxData[1], i_In23 => aTxData[2], i_In24 => aTxData[3], i_In25 => aTxData[4], i_In26 => aTxData[5], i_In27 => aTxData[6], i_In28 => aTxData[7]);
Mov8INT_4(EN := Mov8INT_3.ENO, i_In11 := H0300, i_In12 := H0006, i_In13 := H0000, i_In14 := H0400, i_In15 := H00C8, i_In16 := H00C8, i_In17 := H00A0, i_In18 := 0, i_In21 => aTxData[8], i_In22 => aTxData[9], i_In23 => aTxData[10], i_In24 => aTxData[11], i_In25 => aTxData[12], i_In26 => aTxData[13], i_In27 => aTxData[14], i_In28 => aTxData[15]);
(* network 6 *)
(* CPU 송신 프로그램 Active *)
_e1 := SP_SOCSND(LDP(TRUE, sb50ms) AND SD1288.A AND SD1282.2, U0, 3, acSendDataC, aTxData[0], abSendResC);
INCP(_e1, iVar2);
(* network 7 *)
INC(abSendResC[0] AND NOT abSendResC[1], CntSend1);
_e1 := MOVE_E(abSendResC[0] AND abSendResC[1], acSendDataC[1], ErrCodeSC);
SET(_e1, bSendErrC);
(* network 8 *)
(* CPU 수신 프로그램 Active *)
_e1 := SP_SOCRCV(SD1286.2 AND SD1288.A, U0, 3, acRecvDataC, aRxData[0], abRecvResC);
INCP(_e1, iVar3);
TON_1(IN := NOT SD1286.2, PT := T#5s);
_e2 := INCP(TON_1.Q, CntRecvErr1);
bRecvErrC := _e2;
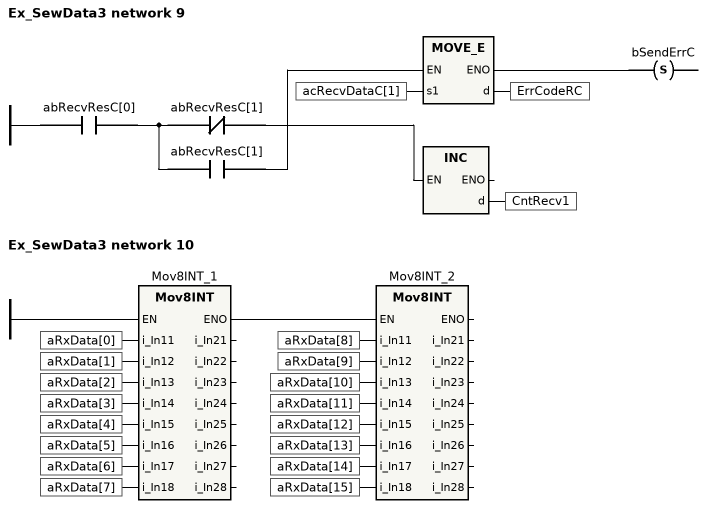
(* network 9 *)
INC(abRecvResC[0] AND NOT abRecvResC[1], CntRecv1);
_e1 := MOVE_E(abRecvResC[0] AND abRecvResC[1], acRecvDataC[1], ErrCodeRC);
SET(_e1, bSendErrC);
(* network 10 *)
Mov8INT_1(EN := TRUE, i_In11 := aRxData[0], i_In12 := aRxData[1], i_In13 := aRxData[2], i_In14 := aRxData[3], i_In15 := aRxData[4], i_In16 := aRxData[5], i_In17 := aRxData[6], i_In18 := aRxData[7]);
Mov8INT_2(EN := Mov8INT_1.ENO, i_In11 := aRxData[8], i_In12 := aRxData[9], i_In13 := aRxData[10], i_In14 := aRxData[11], i_In15 := aRxData[12], i_In16 := aRxData[13], i_In17 := aRxData[14], i_In18 := aRxData[15]);
END_PROGRAM

FUNCTION_BLOCK SewModbus
VAR_INPUT
  Conn : INT;
  CntWord : INT;
END_VAR
VAR_OUTPUT
  bOK : BOOL;
END_VAR
VAR_INPUT
  POdata : ARRAY [0..9] OF INT;
END_VAR
VAR_OUTPUT
  PIdata : ARRAY [0..9] OF INT;
  ErrCode : INT;
END_VAR
VAR_INPUT
  bAct : BOOL;
END_VAR
VAR
  ix : INT;
  iy : INT;
  wMask : WORD;
  aSndData : ARRAY [0..99] OF INT;
  aRcvData : ARRAY [0..99] OF INT;
  bCondOpen : BOOL;
  abOpenRes : ARRAY [0..1] OF BOOL;
  acOpenData : ARRAY [0..9] OF INT;
  bPortOK : BOOL;
  bOpenComp : BOOL;
  bOpenReq : BOOL;
  bRxRecv : BOOL;
  aByteData : ARRAY [0..99] OF INT;
  abCloseRes : ARRAY [0..1] OF BOOL;
  acCloseData : ARRAY [0..1] OF INT;
  abSendRes : ARRAY [0..1] OF BOOL;
  acSendData : ARRAY [0..1] OF INT;
  abRecvRes : ARRAY [0..1] OF BOOL;
  acRecvData : ARRAY [0..1] OF INT;
  iz : INT;
  bCondClose : BOOL;
  bCondSend : BOOL;
  bCondRecv : BOOL;
END_VAR
VAR_OUTPUT
  bRX : BOOL;
END_VAR
;
BSET(TRUE, Conn-1, wMask);
bPortOK 			:= SD1288.A;
bOpenComp	:= (SD1282 AND wMask) <> 0;
bOpenReq		:= (SD1284 AND wMask) <> 0;
bRxRecv			:= (SD1286 AND wMask) <> 0;

(* Open *)
bCondOpen := SM403 AND bPortOK AND NOT bOpenReq AND NOT bOpenComp;
acOpenData[0] := 0;
SP_SOCOPEN(bCondOpen, U0, Conn, acOpenData, abOpenRes);
IF abOpenRes[0] THEN
	IF abOpenRes[1] THEN
		ErrCode := acOpenData[1];
		bOK := FALSE;		 
	ELSE
		bOK := TRUE;		 
	END_IF;
END_IF;

(* Close *)
bCondClose :=  LDF(TRUE, bOpenComp) AND bOpenReq;
SP_SOCCLOSE(bCondClose, U0, Conn, acCloseData, abCloseRes);
IF abCloseRes[0] THEN
	IF abCloseRes[1] THEN
		ErrCode := acCloseData[1];
	END_IF;
END_IF;
 
(* Tx Data *)
bCondSend :=  bPortOK AND bOpenComp AND bAct;
aSndData[0] 		:= CntWord * 2 + 17;
FMOV(TRUE, 0, 50, aByteData[0]);
aByteData[5] 		:= CntWord * 2 + 11;
aByteData[6] 		:= 255;
aByteData[7] 		:= 23;
aByteData[9] 		:= 4;
aByteData[11]	:= CntWord;
aByteData[13]	:= 4;
aByteData[15]	:= CntWord;
aByteData[16]	:= CntWord * 2;
iz := CntWord - 1;
FOR ix := 0 TO iz DO 
	aByteData[17+ix*2]	:= POdata[ix]  / 256; 
	aByteData[18+ix*2]	:= POdata[ix] MOD 256; 
END_FOR;
BTOW(TRUE, aByteData[0], aSndData[0], aSndData[1]);
SP_SOCSND(bCondSend, U0, Conn, acSendData, aSndData[0], abSendRes);
IF abSendRes[0] THEN
	IF abSendRes[1] THEN
		ErrCode := acSendData[1];
	END_IF;
END_IF;

(* Rx Data *)
bCondRecv :=  bPortOK AND bRxRecv;
SP_SOCRCV(bCondRecv, U0, Conn, acRecvData, aRcvData[0], abRecvRes);
IF abRecvRes[0] THEN
	IF abRecvRes[1] THEN
		ErrCode := acRecvData[1];
		bRX := FALSE;
	ELSE
		iy := (aRcvData[0] + 1) / 2;
		FMOV(TRUE, 0, 50, aByteData[0]);
		WTOB(TRUE, aRcvData[1], aRcvData[0], aByteData[0]);	
		ix := aByteData[7];
		IF ix = 23 THEN
			ErrCode := 0;
			bRX := TRUE;
			iz := (aByteData[8] / 2) - 1;
			FOR ix := 0 TO iz DO 
				PIdata[ix] := aByteData[ix*2+9] * 256 + aByteData[ix*2+10];
			END_FOR;
		ELSE
			bRX := FALSE;
			ErrCode := aByteData[8];
		END_IF;
	END_IF;
END_IF;
END_FUNCTION_BLOCK

PROGRAM Ex_SewFC43
VAR
  bOpenReqC : BOOL;
  bCsetReq : BOOL;
  bOpenReqE : BOOL;
  bOpenOkC : BOOL;
  bOpenOkE : BOOL;
  bOpenErrC : BOOL;
  bOpenErrE : BOOL;
  abOpenResC : ARRAY [0..1] OF BOOL;
  abOpenResE : ARRAY [0..1] OF BOOL;
  acOpenData : ARRAY [0..9] OF INT;
  acCsetData : ARRAY [0..4] OF INT;
  acRdCtrl : ARRAY [0..9] OF INT;
  bSendReqC : BOOL;
  bSendReqE : BOOL;
  bSendOkC : BOOL;
  bSendOkE : BOOL;
  bSendErrC : BOOL;
  bSendErrE : BOOL;
  abSendResC : ARRAY [0..1] OF BOOL;
  abSendResE : ARRAY [0..1] OF BOOL;
  abSendResF : ARRAY [0..1] OF BOOL;
  acSendDataC : ARRAY [0..1] OF INT;
  acSendDataE : ARRAY [0..1] OF INT;
  acSendDataF : ARRAY [0..1] OF INT;
  bRecvOkC : BOOL;
  bRecvOkE : BOOL;
  bRecvOkF : BOOL;
  bRecvErrC : BOOL;
  bRecvErrE : BOOL;
  bRecvErrF : BOOL;
  abRecvResC : ARRAY [0..1] OF BOOL;
  abRecvResE : ARRAY [0..1] OF BOOL;
  abRecvResF : ARRAY [0..1] OF BOOL;
  acRecvDataC : ARRAY [0..1] OF INT;
  acRecvDataE : ARRAY [0..1] OF INT;
  acRecvDataF : ARRAY [0..1] OF INT;
  bCloseReq : BOOL;
  bCloseOkC : BOOL;
  bCloseOkE : BOOL;
  bCloseErrC : BOOL;
  bCloseErrE : BOOL;
  abCloseResC : ARRAY [0..1] OF BOOL;
  abCloseResE : ARRAY [0..1] OF BOOL;
  acCloseData : ARRAY [0..1] OF INT;
  CntSend1 : INT;
  CntSend2 : INT;
  CntSend3 : INT;
  CntRecv1 : INT;
  CntRecvErr1 : INT;
  CntRecv2 : INT;
  CntRecv3 : INT;
  CntRecvErr2 : INT;
  CntRecvErr3 : INT;
  ErrCodeSC : INT;
  ErrCodeSE : INT;
  ErrCodeSF : INT;
  ErrCodeRC : INT;
  ErrCodeRE : INT;
  ErrCodeRF : INT;
  Mov4INT_1 : Mov4INT;
  Mov8INT_1 : Mov8INT;
  Mov4INT_2 : Mov4INT;
  Mov4INT_3 : Mov4INT;
  Mov4INT_4 : Mov4INT;
  Word2Bit8_1 : Word2Bit8;
  Word2Bit8_2 : Word2Bit8;
  Word2Bit8_3 : Word2Bit8;
  Word2Bit8_4 : Word2Bit8;
  Word2Bit8_5 : Word2Bit8;
  Word2Bit8_6 : Word2Bit8;
  TON_1 : TON;
  TON_2 : TON;
  TON_3 : TON;
  sbTxReq : BOOL;
  Mov4INT_5 : Mov4INT;
  Mov8INT_2 : Mov8INT;
  Mov8INT_3 : Mov8INT;
  Mov8INT_4 : Mov8INT;
  Mov8INT_5 : Mov8INT;
  TxSet : BOOL;
  TxReq : BOOL;
END_VAR
(* structured ladder/FBD written out as ST: instructions are called as NAME(EN, inputs, outputs); _pN, _eN, _tN stand for wires *)
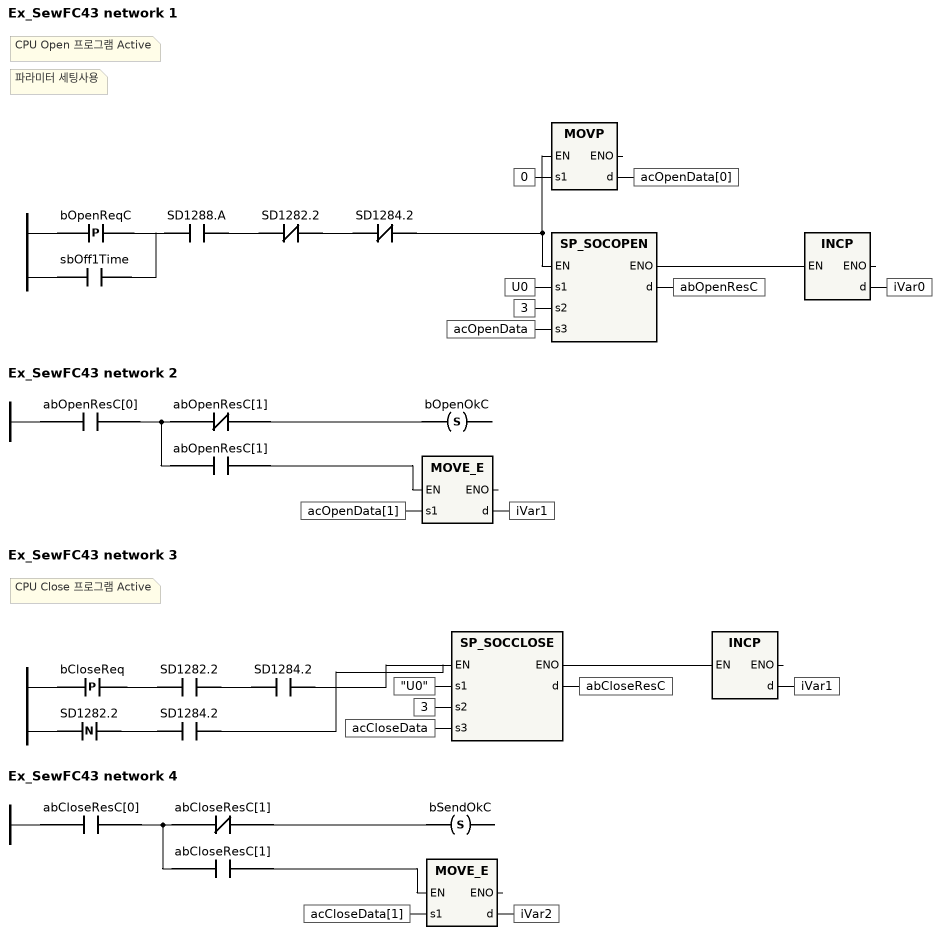
(* network 1 *)
(* CPU Open 프로그램 Active *)
(* 파라미터 세팅사용 *)
_p1 := (((LDP(TRUE, bOpenReqC) OR sbOff1Time) AND SD1288.A) AND NOT SD1282.2) AND NOT SD1284.2;
MOVP(_p1, 0, acOpenData[0]);
_e2 := SP_SOCOPEN(_p1, U0, 3, acOpenData, abOpenResC);
INCP(_e2, iVar0);
(* network 2 *)
SET(abOpenResC[0] AND NOT abOpenResC[1], bOpenOkC);
MOVE_E(abOpenResC[0] AND abOpenResC[1], acOpenData[1], iVar1);
(* network 3 *)
(* CPU Close 프로그램 Active *)
_e1 := SP_SOCCLOSE((LDP(TRUE, bCloseReq) AND SD1282.2 AND SD1284.2) OR (LDF(TRUE, SD1282.2) AND SD1284.2), "U0", 3, acCloseData, abCloseResC);
INCP(_e1, iVar1);
(* network 4 *)
SET(abCloseResC[0] AND NOT abCloseResC[1], bSendOkC);
MOVE_E(abCloseResC[0] AND abCloseResC[1], acCloseData[1], iVar2);
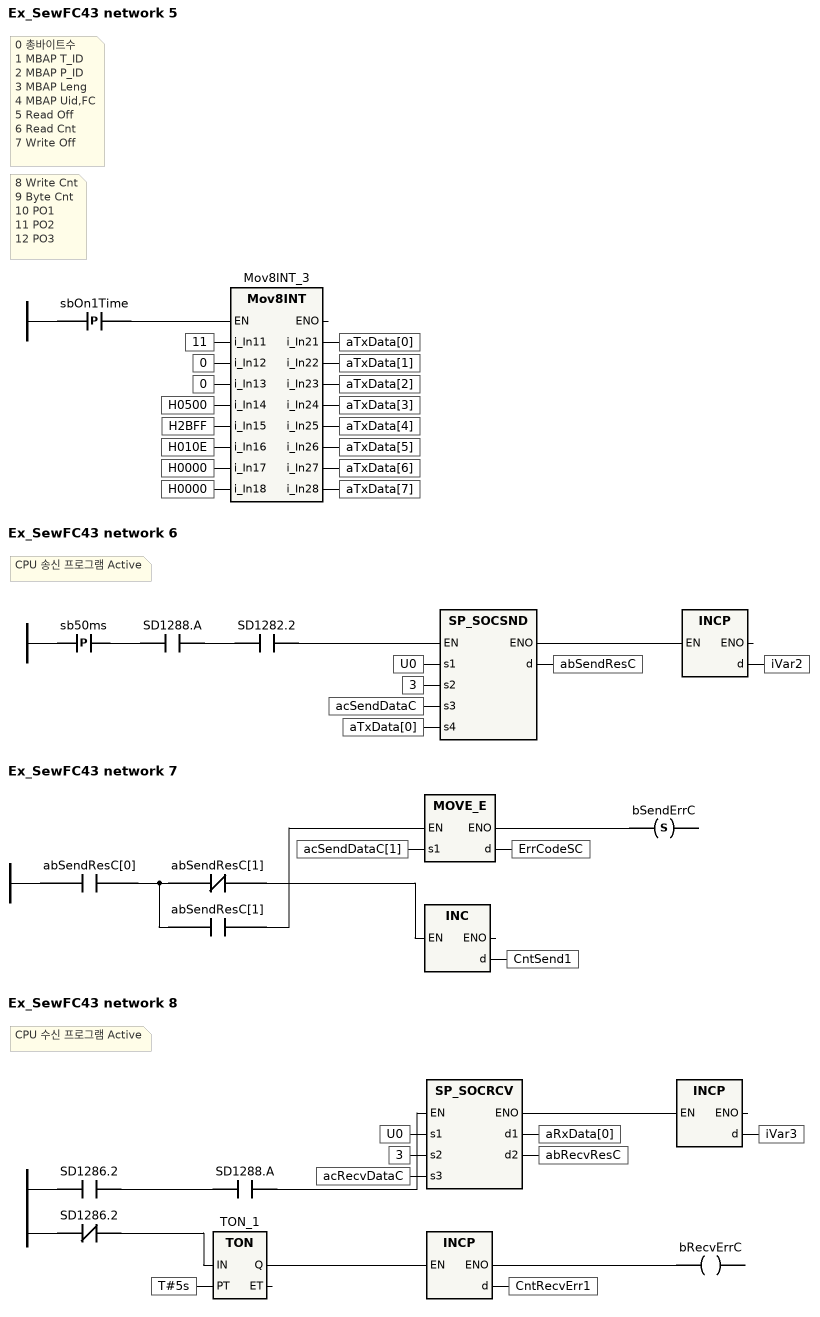
(* network 5 *)
(* 0 총바이트수 / 1 MBAP T_ID / 2 MBAP P_ID / 3 MBAP Leng / 4 MBAP Uid,FC / 5 Read Off / 6 Read Cnt / 7 Write Off *)
(* 8 Write Cnt / 9 Byte Cnt  / 10 PO1 / 11 PO2 / 12 PO3 *)
Mov8INT_3(EN := LDP(TRUE, sbOn1Time), i_In11 := 11, i_In12 := 0, i_In13 := 0, i_In14 := H0500, i_In15 := H2BFF, i_In16 := H010E, i_In17 := H0000, i_In18 := H0000, i_In21 => aTxData[0], i_In22 => aTxData[1], i_In23 => aTxData[2], i_In24 => aTxData[3], i_In25 => aTxData[4], i_In26 => aTxData[5], i_In27 => aTxData[6], i_In28 => aTxData[7]);
(* network 6 *)
(* CPU 송신 프로그램 Active *)
_e1 := SP_SOCSND(LDP(TRUE, sb50ms) AND SD1288.A AND SD1282.2, U0, 3, acSendDataC, aTxData[0], abSendResC);
INCP(_e1, iVar2);
(* network 7 *)
INC(abSendResC[0] AND NOT abSendResC[1], CntSend1);
_e1 := MOVE_E(abSendResC[0] AND abSendResC[1], acSendDataC[1], ErrCodeSC);
SET(_e1, bSendErrC);
(* network 8 *)
(* CPU 수신 프로그램 Active *)
_e1 := SP_SOCRCV(SD1286.2 AND SD1288.A, U0, 3, acRecvDataC, aRxData[0], abRecvResC);
INCP(_e1, iVar3);
TON_1(IN := NOT SD1286.2, PT := T#5s);
_e2 := INCP(TON_1.Q, CntRecvErr1);
bRecvErrC := _e2;
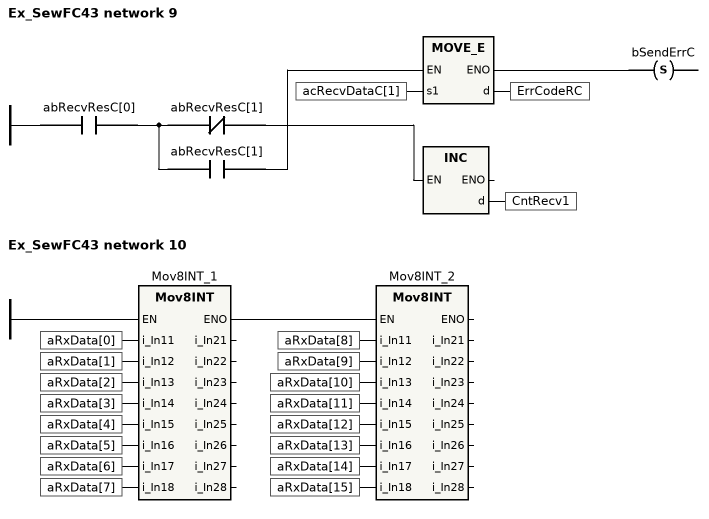
(* network 9 *)
INC(abRecvResC[0] AND NOT abRecvResC[1], CntRecv1);
_e1 := MOVE_E(abRecvResC[0] AND abRecvResC[1], acRecvDataC[1], ErrCodeRC);
SET(_e1, bSendErrC);
(* network 10 *)
Mov8INT_1(EN := TRUE, i_In11 := aRxData[0], i_In12 := aRxData[1], i_In13 := aRxData[2], i_In14 := aRxData[3], i_In15 := aRxData[4], i_In16 := aRxData[5], i_In17 := aRxData[6], i_In18 := aRxData[7]);
Mov8INT_2(EN := Mov8INT_1.ENO, i_In11 := aRxData[8], i_In12 := aRxData[9], i_In13 := aRxData[10], i_In14 := aRxData[11], i_In15 := aRxData[12], i_In16 := aRxData[13], i_In17 := aRxData[14], i_In18 := aRxData[15]);
END_PROGRAM

PROGRAM Ex_Modbus
VAR
  Word2Bit16_1 : Word2Bit16;
  Word2Bit16_2 : Word2Bit16;
  Mov8INT_1 : Mov8INT;
  Mov8INT_2 : Mov8INT;
  aStsD : ARRAY [0..9] OF INT;
  aProcD : ARRAY [0..9] OF INT;
  SewModbus_1 : SewModbus;
  bEnable : BOOL;
  bChange : BOOL;
  wProcD : WORD;
  wStsD : WORD;
END_VAR
(* structured ladder/FBD written out as ST: instructions are called as NAME(EN, inputs, outputs); _pN, _eN, _tN stand for wires *)
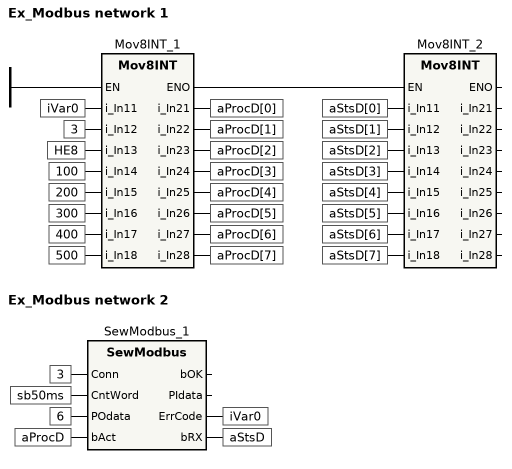
(* network 1 *)
Mov8INT_1(EN := TRUE, i_In11 := iVar0, i_In12 := 3, i_In13 := HE8, i_In14 := 100, i_In15 := 200, i_In16 := 300, i_In17 := 400, i_In18 := 500, i_In21 => aProcD[0], i_In22 => aProcD[1], i_In23 => aProcD[2], i_In24 => aProcD[3], i_In25 => aProcD[4], i_In26 => aProcD[5], i_In27 => aProcD[6], i_In28 => aProcD[7]);
Mov8INT_2(EN := Mov8INT_1.ENO, i_In11 := aStsD[0], i_In12 := aStsD[1], i_In13 := aStsD[2], i_In14 := aStsD[3], i_In15 := aStsD[4], i_In16 := aStsD[5], i_In17 := aStsD[6], i_In18 := aStsD[7]);
(* network 2 *)
SewModbus_1(Conn := 3, CntWord := sb50ms, POdata := 6, bAct := aProcD, ErrCode => iVar0, bRX => aStsD);
END_PROGRAM

PROGRAM Ex_StartMT91
VAR
  Mov8INT_1 : Mov8INT;
  Mov8INT_2 : Mov8INT;
  aStsD : ARRAY [0..9] OF INT;
  aProcD : ARRAY [0..9] OF INT;
END_VAR
(* structured ladder/FBD written out as ST: instructions are called as NAME(EN, inputs, outputs); _pN, _eN, _tN stand for wires *)
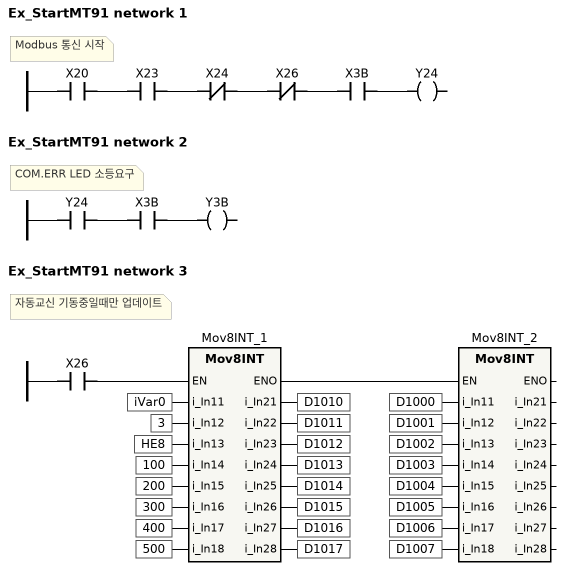
(* network 1 *)
(* Modbus 통신 시작 *)
Y24 := X20 AND X23 AND NOT X24 AND NOT X26 AND X3B;
(* network 2 *)
(* COM.ERR LED 소등요구 *)
Y3B := Y24 AND X3B;
(* network 3 *)
(* 자동교신 기동중일때만 업데이트 *)
Mov8INT_1(EN := X26, i_In11 := iVar0, i_In12 := 3, i_In13 := HE8, i_In14 := 100, i_In15 := 200, i_In16 := 300, i_In17 := 400, i_In18 := 500, i_In21 => D1010, i_In22 => D1011, i_In23 => D1012, i_In24 => D1013, i_In25 => D1014, i_In26 => D1015, i_In27 => D1016, i_In28 => D1017);
Mov8INT_2(EN := Mov8INT_1.ENO, i_In11 := D1000, i_In12 := D1001, i_In13 := D1002, i_In14 := D1003, i_In15 := D1004, i_In16 := D1005, i_In17 := D1006, i_In18 := D1007);
END_PROGRAM

PROGRAM EyEthREAD_WRITE
(* structured ladder/FBD written out as ST: instructions are called as NAME(EN, inputs, outputs); _pN, _eN, _tN stand for wires *)
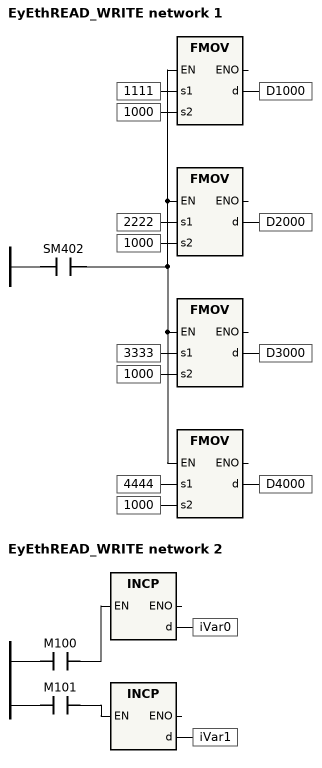
(* network 1 *)
FMOV(SM402, 1111, 1000, D1000);
FMOV(SM402, 2222, 1000, D2000);
FMOV(SM402, 3333, 1000, D3000);
FMOV(SM402, 4444, 1000, D4000);
(* network 2 *)
INCP(M100, iVar0);
INCP(M101, iVar1);
END_PROGRAM

PROGRAM Ex_CmdMT91
VAR
  Mov8INT_1 : Mov8INT;
  Mov8INT_2 : Mov8INT;
  aStsD : ARRAY [0..9] OF INT;
  aProcD : ARRAY [0..9] OF INT;
  bErr1 : BOOL;
  ErrCode1 : INT;
END_VAR
(* structured ladder/FBD written out as ST: instructions are called as NAME(EN, inputs, outputs); _pN, _eN, _tN stand for wires *)
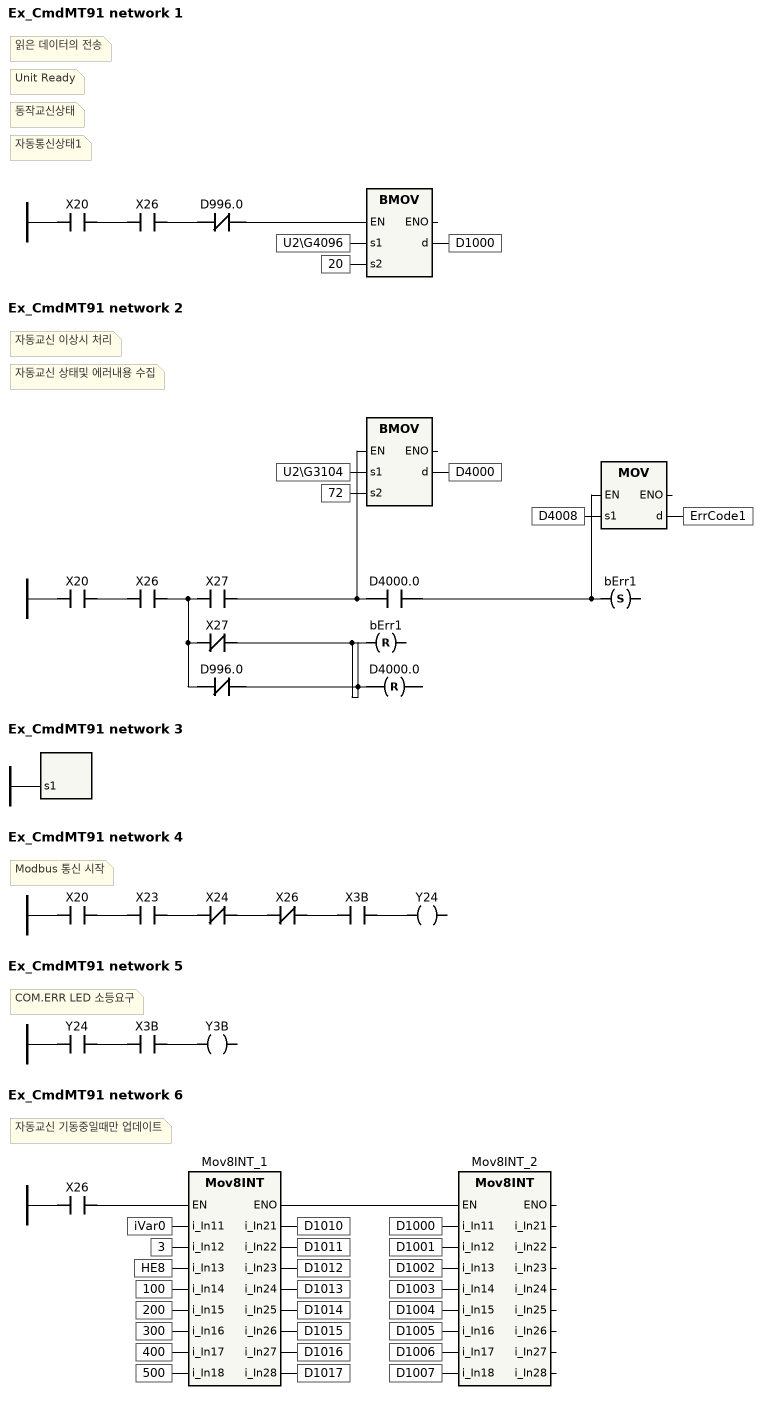
(* network 1 *)
(* 읽은 데이터의 전송 *)
(* Unit Ready *)
(* 동작교신상태 *)
(* 자동통신상태1 *)
BMOV(X20 AND X26 AND NOT D996.0, U2\G4096, 20, D1000);
(* network 2 *)
(* 자동교신 이상시 처리 *)
(* 자동교신 상태및 에러내용 수집 *)
_p1 := X20 AND X26;
_p2 := _p1 AND X27;
BMOV(_p2, U2\G3104, 72, D4000);
_p3 := _p2 AND D4000.0;
SET(_p3, bErr1);
MOV(_p3, D4008, ErrCode1);
_p4 := (_p1 AND NOT X27) OR (_p1 AND NOT D996.0);
RST(_p4, bErr1);
RST(_p4, D4000.0);
(* network 3 *)
(* element kind 10  <- TRUE *)
(* network 4 *)
(* Modbus 통신 시작 *)
Y24 := X20 AND X23 AND NOT X24 AND NOT X26 AND X3B;
(* network 5 *)
(* COM.ERR LED 소등요구 *)
Y3B := Y24 AND X3B;
(* network 6 *)
(* 자동교신 기동중일때만 업데이트 *)
Mov8INT_1(EN := X26, i_In11 := iVar0, i_In12 := 3, i_In13 := HE8, i_In14 := 100, i_In15 := 200, i_In16 := 300, i_In17 := 400, i_In18 := 500, i_In21 => D1010, i_In22 => D1011, i_In23 => D1012, i_In24 => D1013, i_In25 => D1014, i_In26 => D1015, i_In27 => D1016, i_In28 => D1017);
Mov8INT_2(EN := Mov8INT_1.ENO, i_In11 := D1000, i_In12 := D1001, i_In13 := D1002, i_In14 := D1003, i_In15 := D1004, i_In16 := D1005, i_In17 := D1006, i_In18 := D1007);
END_PROGRAM

PROGRAM ExSEND_RECV
VAR
  Mov8INT_1 : Mov8INT;
  acSndCtrl : ARRAY [0..17] OF INT;
  abSndComp : ARRAY [0..1] OF BOOL;
  aSndData : ARRAY [0..3] OF INT;
  Mov8INT_2 : Mov8INT;
  aAnsData : ARRAY [0..5] OF INT;
  Mov4INT_1 : Mov4INT;
  iCntSndOk : INT;
  iCntSndErr : INT;
  acRevCtrl : ARRAY [0..17] OF INT;
  abRevComp : ARRAY [0..1] OF BOOL;
  iCntRevOk : INT;
  iCntRevErr : INT;
  Mov4INT_2 : Mov4INT;
  aRevData : ARRAY [0..3] OF INT;
  Mov4INT_3 : Mov4INT;
  Mov4INT_4 : Mov4INT;
  SendCmd : BOOL;
  RecvCmd : BOOL;
END_VAR
(* structured ladder/FBD written out as ST: instructions are called as NAME(EN, inputs, outputs); _pN, _eN, _tN stand for wires *)
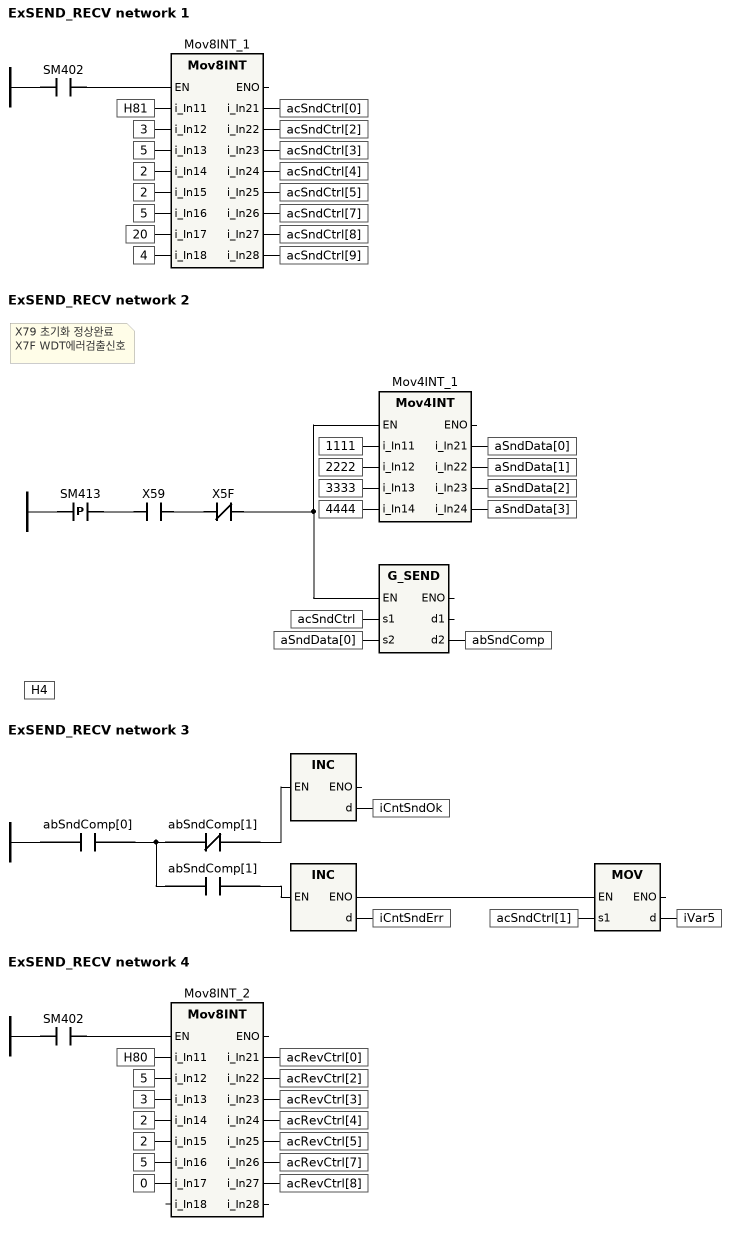
(* network 1 *)
Mov8INT_1(EN := SM402, i_In11 := H81, i_In12 := 3, i_In13 := 5, i_In14 := 2, i_In15 := 2, i_In16 := 5, i_In17 := 20, i_In18 := 4, i_In21 => acSndCtrl[0], i_In22 => acSndCtrl[2], i_In23 => acSndCtrl[3], i_In24 => acSndCtrl[4], i_In25 => acSndCtrl[5], i_In26 => acSndCtrl[7], i_In27 => acSndCtrl[8], i_In28 => acSndCtrl[9]);
(* network 2 *)
(* X79 초기화 정상완료 / X7F WDT에러검출신호 *)
_p1 := LDP(TRUE, SM413) AND X59 AND NOT X5F;
Mov4INT_1(EN := _p1, i_In11 := 1111, i_In12 := 2222, i_In13 := 3333, i_In14 := 4444, i_In21 => aSndData[0], i_In22 => aSndData[1], i_In23 => aSndData[2], i_In24 => aSndData[3]);
G_SEND(_p1, acSndCtrl, aSndData[0], _open, abSndComp);
(* not connected to any output: H4 *)
(* network 3 *)
INC(abSndComp[0] AND NOT abSndComp[1], iCntSndOk);
_e1 := INC(abSndComp[0] AND abSndComp[1], iCntSndErr);
MOV(_e1, acSndCtrl[1], iVar5);
(* network 4 *)
Mov8INT_2(EN := SM402, i_In11 := H80, i_In12 := 5, i_In13 := 3, i_In14 := 2, i_In15 := 2, i_In16 := 5, i_In17 := 0, i_In21 => acRevCtrl[0], i_In22 => acRevCtrl[2], i_In23 => acRevCtrl[3], i_In24 => acRevCtrl[4], i_In25 => acRevCtrl[5], i_In26 => acRevCtrl[7], i_In27 => acRevCtrl[8]);
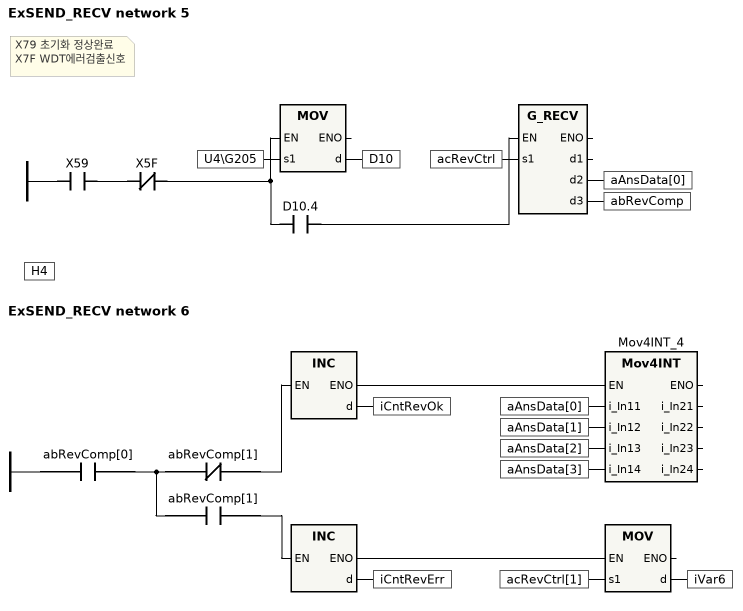
(* network 5 *)
(* X79 초기화 정상완료 / X7F WDT에러검출신호 *)
_p1 := X59 AND NOT X5F;
MOV(_p1, U4\G205, D10);
G_RECV(_p1 AND D10.4, acRevCtrl, _open, aAnsData[0], abRevComp);
(* not connected to any output: H4 *)
(* network 6 *)
_e1 := INC(abRevComp[0] AND NOT abRevComp[1], iCntRevOk);
Mov4INT_4(EN := _e1, i_In11 := aAnsData[0], i_In12 := aAnsData[1], i_In13 := aAnsData[2], i_In14 := aAnsData[3]);
_e2 := INC(abRevComp[0] AND abRevComp[1], iCntRevErr);
MOV(_e2, acRevCtrl[1], iVar6);
END_PROGRAM

PROGRAM ExZNRD_ZNWR
VAR
  Mov8INT_1 : Mov8INT;
  acRdCtrl : ARRAY [0..17] OF INT;
  abRdComp : ARRAY [0..1] OF BOOL;
  iCntRdOk : INT;
  iCntRdErr : INT;
  acWrCtrl : ARRAY [0..17] OF INT;
  abWrComp : ARRAY [0..1] OF BOOL;
  Mov8INT_2 : Mov8INT;
  iCntWrOk : INT;
  iCntWrErr : INT;
END_VAR
(* structured ladder/FBD written out as ST: instructions are called as NAME(EN, inputs, outputs); _pN, _eN, _tN stand for wires *)
